KUKA KRL program: EPS_2_251491_MH02A_A_20251118025154.src

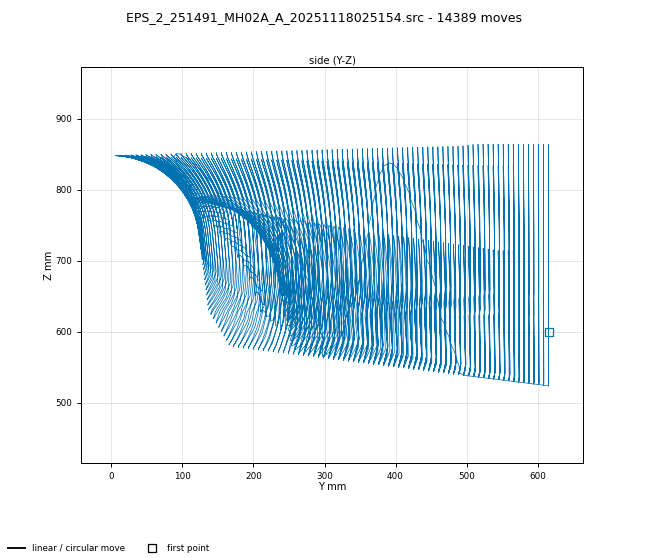
[picture p0: tool path of EPS_2_251491_MH02A_A_20251118025154.src, 14389 of 14391 moves have a stored position in this frame; points joined in program order, loops and branches not executed]
&ACCESS RVP
&REL 4
&COMMENT QRS 19112012
&PARAM EDITMASK = *
DEF PART()
EXT BAS (BAS_COMMAND :IN,REAL :IN )
INT I
BAS (#INITMOV,0 )

;KUKA QRS Post kuka4.cps  Date:22-06-2017 !

File_ID=2920

QRS_PRE_INIT()

;Init var - Until changes are made in qrs_pre_init
Outlet_Square_prg=0
Inlet_1_Square_prg=0
Inlet_2_Square_prg=0
Inlet_3_Square_prg=0
Inlet_4_Square_prg=0
Inlet_5_Square_prg=0

Outlet_1={X 0.000, Y 513.730, Z 763.500, B 0.000, E1 0.000 }
Inlet_1={X 0.000, Y 515.870, Z 733.500, B 0.000, E1 180.000 }
Inlet_2={X 0.000, Y 545.110, Z 323.500, B 0.000, E1 248.000 }
Outlet_1_type=201
Inlet_1_type=201
Inlet_2_type=201
;QRS#1=Sidecore dimensions
;QRS#2=200-8" PVC SDR 35
;QRS#3=200-8" PVC SDR 35
;QRS#4=200-8" PVC SDR 35
;QRS#5=
;QRS#6=
;QRS#7=
;QRS#8=
;QRS#9=12-08 PSX
;QRS#10=12-08 PSX
;QRS#11=12-08 PSX
;QRS#12=
;QRS#13=
;QRS#14=
;QRS#15=
;QRS#16=1220x127x1143 3,75'
;QRS#17=EPS Height
;QRS#18=864
;QRS#19=*
;QRS#20= UPDATED VERSION 22-06-2017
;QRS#21=*
Outlet_Square=0100
Inlet_1_Square=0100
Inlet_2_Square=0100
Inlet_3_Square=0
Inlet_4_Square=0
Inlet_5_Square=0
Mill_Square=1
Outlet_Square_Prg=204
Inlet_1_Square_prg=204
Inlet_2_Square_prg=204

QRS_INIT()

$ADVANCE=5

; T1
PTP {E1 173.604,E2 173.604}
PTP {X 0,Y 615.506,A -85,B 0,C 180,E1 173.604,E2 173.604,E3 0,E4 0,E5 0,E6 0}
QRS_SPEED_INIT()
LIN {X 0,Y 615.506,Z 600,A -85,B 0,C 180,E1 173.604,E2 173.604,E3 0,E4 0,E5 0,E6 0} C_VEL
LIN {X 0,Y 615.506,Z 533.863,A -85,B 0,C 180,E1 173.604,E2 173.604} C_VEL
LIN {X 0,Y 615.506,Z 525.682,A -85,B 0,C 180,E1 173.604,E2 173.604} C_VEL
LIN {X 0,Y 615.488,Z 523.682,A -85,B 0,C 180,E1 173.418,E2 173.418} C_VEL
LIN {X 0,Y 615.475,Z 523.688,A -85,B 0,C 180,E1 170.801,E2 170.801} C_VEL
LIN {X 0,Y 615.491,Z 523.701,A -85,B 0,C 180,E1 168.139,E2 168.139} C_VEL
LIN {X 0,Y 615.482,Z 523.685,A -85,B 0,C 180,E1 165.451,E2 165.451} C_VEL
LIN {X 0,Y 615.476,Z 523.687,A -85,B 0,C 180,E1 162.729,E2 162.729} C_VEL
LIN {X 0,Y 615.49,Z 523.699,A -85,B 0,C 180,E1 159.967,E2 159.967} C_VEL
LIN {X 0,Y 615.487,Z 523.682,A -85,B 0,C 180,E1 157.155,E2 157.155} C_VEL
LIN {X 0,Y 615.484,Z 523.693,A -85,B 0,C 180,E1 154.284,E2 154.284} C_VEL
LIN {X 0,Y 615.48,Z 523.691,A -85,B 0,C 180,E1 151.551,E2 151.551} C_VEL
LIN {X 0,Y 615.484,Z 523.682,A -85,B 0,C 180,E1 148.914,E2 148.914} C_VEL
LIN {X 0,Y 615.496,Z 523.697,A -85,B 0,C 180,E1 145.978,E2 145.978} C_VEL
LIN {X 0,Y 615.487,Z 523.682,A -85,B 0,C 180,E1 143.063,E2 143.063} C_VEL
LIN {X 0,Y 615.477,Z 523.691,A -85,B 0,C 180,E1 140.249,E2 140.249} C_VEL
LIN {X 0,Y 615.489,Z 523.697,A -85,B 0,C 180,E1 137.647,E2 137.647} C_VEL
LIN {X 0,Y 615.479,Z 523.684,A -85,B 0,C 180,E1 134.93,E2 134.93} C_VEL
LIN {X 0,Y 615.478,Z 523.692,A -85,B 0,C 180,E1 132.079,E2 132.079} C_VEL
LIN {X 0,Y 615.494,Z 523.699,A -85,B 0,C 180,E1 129.75,E2 129.75} C_VEL
LIN {X 0,Y 615.478,Z 523.685,A -85,B 0,C 180,E1 126.935,E2 126.935} C_VEL
LIN {X 0,Y 615.489,Z 523.681,A -85,B 0,C 180,E1 124.7,E2 124.7} C_VEL
LIN {X 0,Y 615.485,Z 523.683,A -85,B 0,C 180,E1 122.33,E2 122.33} C_VEL
LIN {X 0,Y 615.493,Z 523.696,A -85,B 0,C 180,E1 119.406,E2 119.406} C_VEL
LIN {X 0,Y 615.492,Z 523.68,A -85,B 0,C 180,E1 116.444,E2 116.444} C_VEL
LIN {X 0,Y 615.488,Z 523.846,A -85,B 0,C 180,E1 114.239,E2 114.239} C_VEL
LIN {X 0,Y 615.492,Z 547.088,A -85,B 0,C 180,E1 111.432,E2 111.432} C_VEL
LIN {X 0,Y 615.493,Z 570.943,A -85,B 0,C 180,E1 108.605,E2 108.605} C_VEL
LIN {X 0,Y 615.486,Z 594.072,A -85,B 0,C 180,E1 105.906,E2 105.906} C_VEL
LIN {X 0,Y 615.486,Z 618.987,A -85,B 0,C 180,E1 103.034,E2 103.034} C_VEL
LIN {X 0,Y 615.479,Z 620.636,A -85,B 0,C 180,E1 102.845,E2 102.845} C_VEL
LIN {X 0,Y 615.476,Z 729.625,A -85,B 0,C 180,E1 101.548,E2 101.548} C_VEL
LIN {X 0,Y 615.49,Z 742.21,A -85,B 0,C 180,E1 101.277,E2 101.277} C_VEL
LIN {X 0,Y 615.489,Z 755.605,A -85,B 0,C 180,E1 100.842,E2 100.842} C_VEL
LIN {X 0,Y 615.493,Z 766.557,A -85,B 0,C 180,E1 100.361,E2 100.361} C_VEL
LIN {X 0,Y 615.485,Z 778.299,A -85,B 0,C 180,E1 99.697,E2 99.697} C_VEL
LIN {X 0,Y 615.499,Z 788.762,A -85,B 0,C 180,E1 98.951,E2 98.951} C_VEL
LIN {X 0,Y 615.498,Z 797.326,A -85,B 0,C 180,E1 98.206,E2 98.206} C_VEL
LIN {X 0,Y 615.497,Z 805.205,A -85,B 0,C 180,E1 97.381,E2 97.381} C_VEL
LIN {X 0,Y 615.497,Z 812.896,A -85,B 0,C 180,E1 96.392,E2 96.392} C_VEL
LIN {X 0,Y 615.497,Z 819.955,A -85,B 0,C 180,E1 95.242,E2 95.242} C_VEL
LIN {X 0,Y 615.494,Z 824.656,A -85,B 0,C 180,E1 94.257,E2 94.257} C_VEL
LIN {X 0,Y 615.494,Z 828.253,A -85,B 0,C 180,E1 93.273,E2 93.273} C_VEL
LIN {X 0,Y 615.496,Z 830.113,A -85,B 0,C 180,E1 92.618,E2 92.618} C_VEL
LIN {X 0,Y 615.497,Z 831.533,A -85,B 0,C 180,E1 91.964,E2 91.964} C_VEL
LIN {X 0,Y 615.496,Z 833.141,A -85,B 0,C 180,E1 90.655,E2 90.655} C_VEL
LIN {X 0,Y 615.495,Z 833.384,A -85,B 0,C 180,E1 90.001,E2 90.001} C_VEL
LIN {X 0,Y 615.495,Z 833.206,A -85,B 0,C 180,E1 89.346,E2 89.346} C_VEL
LIN {X 0,Y 615.498,Z 831.683,A -85,B 0,C 180,E1 88.038,E2 88.038} C_VEL
LIN {X 0,Y 615.498,Z 830.343,A -85,B 0,C 180,E1 87.383,E2 87.383} C_VEL
LIN {X 0,Y 615.496,Z 827.496,A -85,B 0,C 180,E1 86.4,E2 86.4} C_VEL
LIN {X 0,Y 615.498,Z 823.637,A -85,B 0,C 180,E1 85.416,E2 85.416} C_VEL
LIN {X 0,Y 615.498,Z 818.655,A -85,B 0,C 180,E1 84.431,E2 84.431} C_VEL
LIN {X 0,Y 615.496,Z 812.208,A -85,B 0,C 180,E1 83.418,E2 83.418} C_VEL
LIN {X 0,Y 615.497,Z 804.543,A -85,B 0,C 180,E1 82.455,E2 82.455} C_VEL
LIN {X 0,Y 615.498,Z 794.766,A -85,B 0,C 180,E1 81.464,E2 81.464} C_VEL
LIN {X 0,Y 615.497,Z 784.503,A -85,B 0,C 180,E1 80.636,E2 80.636} C_VEL
LIN {X 0,Y 615.496,Z 772.941,A -85,B 0,C 180,E1 79.89,E2 79.89} C_VEL
LIN {X 0,Y 615.496,Z 761.057,A -85,B 0,C 180,E1 79.292,E2 79.292} C_VEL
LIN {X 0,Y 615.497,Z 748.181,A -85,B 0,C 180,E1 78.808,E2 78.808} C_VEL
LIN {X 0,Y 615.477,Z 735.593,A -85,B 0,C 180,E1 78.474,E2 78.474} C_VEL
LIN {X 0,Y 615.475,Z 722.503,A -85,B 0,C 180,E1 78.265,E2 78.265} C_VEL
LIN {X 0,Y 615.48,Z 621.405,A -85,B 0,C 180,E1 77.072,E2 77.072} C_VEL
LIN {X 0,Y 615.476,Z 599.659,A -85,B 0,C 180,E1 74.265,E2 74.265} C_VEL
LIN {X 0,Y 615.487,Z 578.943,A -85,B 0,C 180,E1 71.56,E2 71.56} C_VEL
LIN {X 0,Y 615.485,Z 557.708,A -85,B 0,C 180,E1 68.745,E2 68.745} C_VEL
LIN {X 0,Y 615.476,Z 537.338,A -85,B 0,C 180,E1 65.995,E2 65.995} C_VEL
LIN {X 0,Y 615.474,Z 523.686,A -85,B 0,C 180,E1 64.103,E2 64.103} C_VEL
LIN {X 0,Y 615.485,Z 523.686,A -85,B 0,C 180,E1 61.343,E2 61.343} C_VEL
LIN {X 0,Y 615.492,Z 523.696,A -85,B 0,C 180,E1 58.914,E2 58.914} C_VEL
LIN {X 0,Y 615.497,Z 523.69,A -85,B 0,C 180,E1 56.465,E2 56.465} C_VEL
LIN {X 0,Y 615.48,Z 523.684,A -85,B 0,C 180,E1 53.576,E2 53.576} C_VEL
LIN {X 0,Y 615.488,Z 523.694,A -85,B 0,C 180,E1 50.938,E2 50.938} C_VEL
LIN {X 0,Y 615.496,Z 523.695,A -85,B 0,C 180,E1 48.528,E2 48.528} C_VEL
LIN {X 0,Y 615.477,Z 523.685,A -85,B 0,C 180,E1 45.851,E2 45.851} C_VEL
LIN {X 0,Y 615.493,Z 523.688,A -85,B 0,C 180,E1 43.05,E2 43.05} C_VEL
LIN {X 0,Y 615.493,Z 523.685,A -85,B 0,C 180,E1 40.092,E2 40.092} C_VEL
LIN {X 0,Y 615.489,Z 523.684,A -85,B 0,C 180,E1 37.242,E2 37.242} C_VEL
LIN {X 0,Y 615.497,Z 523.701,A -85,B 0,C 180,E1 34.575,E2 34.575} C_VEL
LIN {X 0,Y 615.474,Z 610.382,A -85,B 0,C 180,E1 33.535,E2 33.535} C_VEL
LIN {X 0,Y 615.48,Z 623.669,A -85,B 0,C 180,E1 33.237,E2 33.237} C_VEL
LIN {X 0,Y 615.494,Z 636.803,A -85,B 0,C 180,E1 32.797,E2 32.797} C_VEL
LIN {X 0,Y 615.482,Z 648.688,A -85,B 0,C 180,E1 32.251,E2 32.251} C_VEL
LIN {X 0,Y 615.486,Z 660.755,A -85,B 0,C 180,E1 31.536,E2 31.536} C_VEL
LIN {X 0,Y 615.497,Z 671.49,A -85,B 0,C 180,E1 30.729,E2 30.729} C_VEL
LIN {X 0,Y 615.499,Z 681.399,A -85,B 0,C 180,E1 29.799,E2 29.799} C_VEL
LIN {X 0,Y 615.497,Z 689.587,A -85,B 0,C 180,E1 28.844,E2 28.844} C_VEL
LIN {X 0,Y 615.493,Z 697.177,A -85,B 0,C 180,E1 27.73,E2 27.73} C_VEL
LIN {X 0,Y 615.493,Z 702.466,A -85,B 0,C 180,E1 26.746,E2 26.746} C_VEL
LIN {X 0,Y 615.496,Z 707.29,A -85,B 0,C 180,E1 25.573,E2 25.573} C_VEL
LIN {X 0,Y 615.493,Z 709.114,A -85,B 0,C 180,E1 24.992,E2 24.992} C_VEL
LIN {X 0,Y 615.494,Z 711.448,A -85,B 0,C 180,E1 24.013,E2 24.013} C_VEL
LIN {X 0,Y 615.496,Z 713.008,A -85,B 0,C 180,E1 22.844,E2 22.844} C_VEL
LIN {X 0,Y 615.495,Z 713.351,A -85,B 0,C 180,E1 22.136,E2 22.136} C_VEL
LIN {X 0,Y 615.497,Z 713.263,A -85,B 0,C 180,E1 21.432,E2 21.432} C_VEL
LIN {X 0,Y 615.495,Z 712.482,A -85,B 0,C 180,E1 20.563,E2 20.563} C_VEL
LIN {X 0,Y 615.494,Z 710.235,A -85,B 0,C 180,E1 19.338,E2 19.338} C_VEL
LIN {X 0,Y 615.497,Z 707.103,A -85,B 0,C 180,E1 18.284,E2 18.284} C_VEL
LIN {X 0,Y 615.496,Z 702.986,A -85,B 0,C 180,E1 17.27,E2 17.27} C_VEL
LIN {X 0,Y 615.497,Z 697.127,A -85,B 0,C 180,E1 16.172,E2 16.172} C_VEL
LIN {X 0,Y 615.496,Z 689.518,A -85,B 0,C 180,E1 15.056,E2 15.056} C_VEL
LIN {X 0,Y 615.498,Z 681.234,A -85,B 0,C 180,E1 14.094,E2 14.094} C_VEL
LIN {X 0,Y 615.499,Z 671.722,A -85,B 0,C 180,E1 13.201,E2 13.201} C_VEL
LIN {X 0,Y 615.486,Z 661.855,A -85,B 0,C 180,E1 12.446,E2 12.446} C_VEL
LIN {X 0,Y 615.492,Z 650.912,A -85,B 0,C 180,E1 11.777,E2 11.777} C_VEL
LIN {X 0,Y 615.491,Z 638.717,A -85,B 0,C 180,E1 11.193,E2 11.193} C_VEL
LIN {X 0,Y 615.495,Z 626.639,A -85,B 0,C 180,E1 10.758,E2 10.758} C_VEL
LIN {X 0,Y 615.483,Z 614.11,A -85,B 0,C 180,E1 10.444,E2 10.444} C_VEL
LIN {X 0,Y 615.476,Z 598.256,A -85,B 0,C 180,E1 10.215,E2 10.215} C_VEL
LIN {X 0,Y 615.493,Z 523.77,A -85,B 0,C 180,E1 9.344,E2 9.344} C_VEL
LIN {X 0,Y 615.489,Z 523.682,A -85,B 0,C 180,E1 6.557,E2 6.557} C_VEL
LIN {X 0,Y 615.477,Z 523.687,A -85,B 0,C 180,E1 3.929,E2 3.929} C_VEL
LIN {X 0,Y 615.496,Z 523.701,A -85,B 0,C 180,E1 1.309,E2 1.309} C_VEL
LIN {X 0,Y 615.488,Z 523.685,A -85,B 0,C 180,E1 -1.309,E2 -1.309} C_VEL
LIN {X 0,Y 615.478,Z 523.685,A -85,B 0,C 180,E1 -3.929,E2 -3.929} C_VEL
LIN {X 0,Y 615.489,Z 523.698,A -85,B 0,C 180,E1 -6.592,E2 -6.592} C_VEL
LIN {X 0,Y 615.479,Z 523.689,A -85,B 0,C 180,E1 -9.199,E2 -9.199} C_VEL
LIN {X 0,Y 615.485,Z 523.682,A -85,B 0,C 180,E1 -11.861,E2 -11.861} C_VEL
LIN {X 0,Y 615.48,Z 523.697,A -85,B 0,C 180,E1 -14.549,E2 -14.549} C_VEL
LIN {X 0,Y 615.476,Z 523.689,A -85,B 0,C 180,E1 -17.271,E2 -17.271} C_VEL
LIN {X 0,Y 615.486,Z 523.684,A -85,B 0,C 180,E1 -20.033,E2 -20.033} C_VEL
LIN {X 0,Y 615.492,Z 523.699,A -85,B 0,C 180,E1 -22.844,E2 -22.844} C_VEL
LIN {X 0,Y 615.484,Z 523.682,A -85,B 0,C 180,E1 -25.716,E2 -25.716} C_VEL
LIN {X 0,Y 615.485,Z 523.692,A -85,B 0,C 180,E1 -28.453,E2 -28.453} C_VEL
LIN {X 0,Y 615.487,Z 523.692,A -85,B 0,C 180,E1 -31.088,E2 -31.088} C_VEL
LIN {X 0,Y 615.496,Z 523.681,A -85,B 0,C 180,E1 -34.022,E2 -34.022} C_VEL
LIN {X 0,Y 615.494,Z 523.697,A -85,B 0,C 180,E1 -36.94,E2 -36.94} C_VEL
LIN {X 0,Y 615.475,Z 523.685,A -85,B 0,C 180,E1 -39.751,E2 -39.751} C_VEL
LIN {X 0,Y 615.493,Z 523.686,A -85,B 0,C 180,E1 -42.353,E2 -42.353} C_VEL
LIN {X 0,Y 615.492,Z 523.694,A -85,B 0,C 180,E1 -45.068,E2 -45.068} C_VEL
LIN {X 0,Y 615.477,Z 523.684,A -85,B 0,C 180,E1 -47.921,E2 -47.921} C_VEL
LIN {X 0,Y 615.493,Z 523.684,A -85,B 0,C 180,E1 -50.252,E2 -50.252} C_VEL
LIN {X 0,Y 615.491,Z 523.695,A -85,B 0,C 180,E1 -53.063,E2 -53.063} C_VEL
LIN {X 0,Y 615.49,Z 523.688,A -85,B 0,C 180,E1 -55.299,E2 -55.299} C_VEL
LIN {X 0,Y 615.484,Z 523.683,A -85,B 0,C 180,E1 -57.67,E2 -57.67} C_VEL
LIN {X 0,Y 615.498,Z 523.69,A -85,B 0,C 180,E1 -60.595,E2 -60.595} C_VEL
LIN {X 0,Y 615.491,Z 523.683,A -85,B 0,C 180,E1 -63.557,E2 -63.557} C_VEL
LIN {X 0,Y 615.474,Z 523.886,A -85,B 0,C 180,E1 -64.08,E2 -64.08} C_VEL
LIN {X 0,Y 615.484,Z 549.311,A -85,B 0,C 180,E1 -66.801,E2 -66.801} C_VEL
LIN {X 0,Y 615.487,Z 575.784,A -85,B 0,C 180,E1 -69.576,E2 -69.576} C_VEL
LIN {X 0,Y 615.49,Z 603.095,A -85,B 0,C 180,E1 -72.388,E2 -72.388} C_VEL
LIN {X 0,Y 615.481,Z 629.946,A -85,B 0,C 180,E1 -75.113,E2 -75.113} C_VEL
LIN {X 0,Y 615.488,Z 649.643,A -85,B 0,C 180,E1 -77.093,E2 -77.093} C_VEL
LIN {X 0,Y 615.476,Z 759.874,A -85,B 0,C 180,E1 -78.411,E2 -78.411} C_VEL
LIN {X 0,Y 615.487,Z 772.371,A -85,B 0,C 180,E1 -78.683,E2 -78.683} C_VEL
LIN {X 0,Y 615.496,Z 785.511,A -85,B 0,C 180,E1 -79.109,E2 -79.109} C_VEL
LIN {X 0,Y 615.484,Z 797.491,A -85,B 0,C 180,E1 -79.64,E2 -79.64} C_VEL
LIN {X 0,Y 615.483,Z 809.007,A -85,B 0,C 180,E1 -80.304,E2 -80.304} C_VEL
LIN {X 0,Y 615.499,Z 819.35,A -85,B 0,C 180,E1 -81.051,E2 -81.051} C_VEL
LIN {X 0,Y 615.497,Z 827.819,A -85,B 0,C 180,E1 -81.795,E2 -81.795} C_VEL
LIN {X 0,Y 615.498,Z 835.612,A -85,B 0,C 180,E1 -82.62,E2 -82.62} C_VEL
LIN {X 0,Y 615.496,Z 843.207,A -85,B 0,C 180,E1 -83.609,E2 -83.609} C_VEL
LIN {X 0,Y 615.498,Z 850.208,A -85,B 0,C 180,E1 -84.76,E2 -84.76} C_VEL
LIN {X 0,Y 615.494,Z 854.854,A -85,B 0,C 180,E1 -85.744,E2 -85.744} C_VEL
LIN {X 0,Y 615.496,Z 858.4,A -85,B 0,C 180,E1 -86.728,E2 -86.728} C_VEL
LIN {X 0,Y 615.497,Z 860.234,A -85,B 0,C 180,E1 -87.383,E2 -87.383} C_VEL
LIN {X 0,Y 615.496,Z 861.609,A -85,B 0,C 180,E1 -88.038,E2 -88.038} C_VEL
LIN {X 0,Y 615.496,Z 863.174,A -85,B 0,C 180,E1 -89.346,E2 -89.346} C_VEL
LIN {X 0,Y 615.494,Z 863.389,A -85,B 0,C 180,E1 -90.001,E2 -90.001} C_VEL
LIN {X 0,Y 615.496,Z 862.579,A -85,B 0,C 180,E1 -91.309,E2 -91.309} C_VEL
LIN {X 0,Y 615.496,Z 861.607,A -85,B 0,C 180,E1 -91.964,E2 -91.964} C_VEL
LIN {X 0,Y 615.497,Z 860.232,A -85,B 0,C 180,E1 -92.618,E2 -92.618} C_VEL
LIN {X 0,Y 615.496,Z 857.348,A -85,B 0,C 180,E1 -93.601,E2 -93.601} C_VEL
LIN {X 0,Y 615.498,Z 853.439,A -85,B 0,C 180,E1 -94.585,E2 -94.585} C_VEL
LIN {X 0,Y 615.499,Z 848.402,A -85,B 0,C 180,E1 -95.57,E2 -95.57} C_VEL
LIN {X 0,Y 615.497,Z 841.869,A -85,B 0,C 180,E1 -96.583,E2 -96.583} C_VEL
LIN {X 0,Y 615.497,Z 834.129,A -85,B 0,C 180,E1 -97.546,E2 -97.546} C_VEL
LIN {X 0,Y 615.498,Z 826.04,A -85,B 0,C 180,E1 -98.372,E2 -98.372} C_VEL
LIN {X 0,Y 615.499,Z 816.162,A -85,B 0,C 180,E1 -99.199,E2 -99.199} C_VEL
LIN {X 0,Y 615.486,Z 804.975,A -85,B 0,C 180,E1 -99.946,E2 -99.946} C_VEL
LIN {X 0,Y 615.483,Z 794.015,A -85,B 0,C 180,E1 -100.527,E2 -100.527} C_VEL
LIN {X 0,Y 615.496,Z 781.425,A -85,B 0,C 180,E1 -101.042,E2 -101.042} C_VEL
LIN {X 0,Y 615.482,Z 769.049,A -85,B 0,C 180,E1 -101.402,E2 -101.402} C_VEL
LIN {X 0,Y 615.475,Z 755.442,A -85,B 0,C 180,E1 -101.653,E2 -101.653} C_VEL
LIN {X 0,Y 615.493,Z 650.529,A -85,B 0,C 180,E1 -102.887,E2 -102.887} C_VEL
LIN {X 0,Y 615.496,Z 625.281,A -85,B 0,C 180,E1 -105.735,E2 -105.735} C_VEL
LIN {X 0,Y 615.488,Z 601.591,A -85,B 0,C 180,E1 -108.441,E2 -108.441} C_VEL
LIN {X 0,Y 615.491,Z 577.301,A -85,B 0,C 180,E1 -111.256,E2 -111.256} C_VEL
LIN {X 0,Y 615.486,Z 554.004,A -85,B 0,C 180,E1 -114.007,E2 -114.007} C_VEL
LIN {X 0,Y 615.492,Z 531.309,A -85,B 0,C 180,E1 -116.745,E2 -116.745} C_VEL
LIN {X 0,Y 615.483,Z 523.683,A -85,B 0,C 180,E1 -117.684,E2 -117.684} C_VEL
LIN {X 0,Y 615.477,Z 523.685,A -85,B 0,C 180,E1 -120.161,E2 -120.161} C_VEL
LIN {X 0,Y 615.487,Z 523.687,A -85,B 0,C 180,E1 -122.458,E2 -122.458} C_VEL
LIN {X 0,Y 615.491,Z 523.695,A -85,B 0,C 180,E1 -124.815,E2 -124.815} C_VEL
LIN {X 0,Y 615.491,Z 523.694,A -85,B 0,C 180,E1 -127.242,E2 -127.242} C_VEL
LIN {X 0,Y 615.477,Z 523.684,A -85,B 0,C 180,E1 -130.088,E2 -130.088} C_VEL
LIN {X 0,Y 615.478,Z 523.685,A -85,B 0,C 180,E1 -132.354,E2 -132.354} C_VEL
LIN {X 0,Y 615.492,Z 523.7,A -85,B 0,C 180,E1 -135.068,E2 -135.068} C_VEL
LIN {X 0,Y 615.49,Z 523.682,A -85,B 0,C 180,E1 -137.919,E2 -137.919} C_VEL
LIN {X 0,Y 615.475,Z 523.684,A -85,B 0,C 180,E1 -140.249,E2 -140.249} C_VEL
LIN {X 0,Y 615.494,Z 523.695,A -85,B 0,C 180,E1 -143.062,E2 -143.062} C_VEL
LIN {X 0,Y 615.495,Z 523.681,A -85,B 0,C 180,E1 -145.978,E2 -145.978} C_VEL
LIN {X 0,Y 615.478,Z 523.683,A -85,B 0,C 180,E1 -148.314,E2 -148.314} C_VEL
LIN {X 0,Y 615.477,Z 523.685,A -85,B 0,C 180,E1 -150.593,E2 -150.593} C_VEL
LIN {X 0,Y 615.489,Z 523.689,A -85,B 0,C 180,E1 -152.954,E2 -152.954} C_VEL
LIN {X 0,Y 615.485,Z 523.691,A -85,B 0,C 180,E1 -155.728,E2 -155.728} C_VEL
LIN {X 0,Y 615.488,Z 523.688,A -85,B 0,C 180,E1 -157.864,E2 -157.864} C_VEL
LIN {X 0,Y 615.476,Z 523.685,A -85,B 0,C 180,E1 -160.662,E2 -160.662} C_VEL
LIN {X 0,Y 615.495,Z 523.699,A -85,B 0,C 180,E1 -163.414,E2 -163.414} C_VEL
LIN {X 0,Y 615.492,Z 523.684,A -85,B 0,C 180,E1 -166.126,E2 -166.126} C_VEL
LIN {X 0,Y 615.476,Z 523.685,A -85,B 0,C 180,E1 -168.807,E2 -168.807} C_VEL
LIN {X 0,Y 615.496,Z 523.696,A -85,B 0,C 180,E1 -171.463,E2 -171.463} C_VEL
LIN {X 0,Y 615.485,Z 523.687,A -85,B 0,C 180,E1 -174.101,E2 -174.101} C_VEL
LIN {X 0,Y 615.481,Z 523.683,A -85,B 0,C 180,E1 -176.727,E2 -176.727} C_VEL
LIN {X 0,Y 615.483,Z 523.692,A -85,B 0,C 180,E1 -179.346,E2 -179.346} C_VEL
LIN {X 0,Y 615.482,Z 523.695,A -85,B 0,C 180,E1 -181.963,E2 -181.963} C_VEL
LIN {X 0,Y 615.498,Z 523.679,A -85,B 0,C 180,E1 -184.585,E2 -184.585} C_VEL
LIN {X 0,Y 615.488,Z 523.682,A -85,B 0,C 180,E1 -186.582,E2 -186.582} C_VEL
LIN {X 0,Y 614.804,Z 523.835,A -85,B 0,C 180,E1 -187.128,E2 -187.128} C_VEL
LIN {X 0,Y 611.96,Z 524.257,A -85,B 0,C 180,E1 -188.014,E2 -188.014} C_VEL
LIN {X 0,Y 609.57,Z 524.564,A -85,B 0,C 180,E1 -188.726,E2 -188.726} C_VEL
LIN {X 0,Y 608.541,Z 524.68,A -85,B 0,C 180,E1 -189.276,E2 -189.276} C_VEL
LIN {X 0,Y 608.456,Z 524.69,A -85,B 0,C 180,E1 -189.462,E2 -189.462} C_VEL
LIN {X 0,Y 608.466,Z 524.693,A -85,B 0,C 180,E1 -192,E2 -192} C_VEL
LIN {X 0,Y 608.47,Z 524.685,A -85,B 0,C 180,E1 -194.721,E2 -194.721} C_VEL
LIN {X 0,Y 608.449,Z 524.691,A -85,B 0,C 180,E1 -197.477,E2 -197.477} C_VEL
LIN {X 0,Y 608.463,Z 524.691,A -85,B 0,C 180,E1 -200.274,E2 -200.274} C_VEL
LIN {X 0,Y 608.448,Z 524.688,A -85,B 0,C 180,E1 -203.124,E2 -203.124} C_VEL
LIN {X 0,Y 608.468,Z 524.691,A -85,B 0,C 180,E1 -205.721,E2 -205.721} C_VEL
LIN {X 0,Y 608.448,Z 524.694,A -85,B 0,C 180,E1 -208.267,E2 -208.267} C_VEL
LIN {X 0,Y 608.474,Z 524.687,A -85,B 0,C 180,E1 -210.545,E2 -210.545} C_VEL
LIN {X 0,Y 608.453,Z 524.687,A -85,B 0,C 180,E1 -212.88,E2 -212.88} C_VEL
LIN {X 0,Y 608.434,Z 524.689,A -85,B 0,C 180,E1 -215.279,E2 -215.279} C_VEL
LIN {X 0,Y 608.472,Z 524.688,A -85,B 0,C 180,E1 -217.746,E2 -217.746} C_VEL
LIN {X 0,Y 608.452,Z 524.696,A -85,B 0,C 180,E1 -220.329,E2 -220.329} C_VEL
LIN {X 0,Y 608.484,Z 524.683,A -85,B 0,C 180,E1 -223.31,E2 -223.31} C_VEL
LIN {X 0,Y 608.466,Z 524.694,A -85,B 0,C 180,E1 -226.13,E2 -226.13} C_VEL
LIN {X 0,Y 608.447,Z 524.69,A -85,B 0,C 180,E1 -228.823,E2 -228.823} C_VEL
LIN {X 0,Y 608.461,Z 524.688,A -85,B 0,C 180,E1 -231.761,E2 -231.761} C_VEL
LIN {X 0,Y 608.449,Z 524.691,A -85,B 0,C 180,E1 -233.955,E2 -233.955} C_VEL
LIN {X 0,Y 608.467,Z 524.695,A -85,B 0,C 180,E1 -236.329,E2 -236.329} C_VEL
LIN {X 0,Y 608.446,Z 524.693,A -85,B 0,C 180,E1 -238.733,E2 -238.733} C_VEL
LIN {X 0,Y 608.474,Z 524.684,A -85,B 0,C 180,E1 -241.38,E2 -241.38} C_VEL
LIN {X 0,Y 608.475,Z 524.692,A -85,B 0,C 180,E1 -244.279,E2 -244.279} C_VEL
LIN {X 0,Y 608.494,Z 524.843,A -85,B 0,C 180,E1 -245.587,E2 -245.587} C_VEL
LIN {X 0,Y 608.637,Z 540.255,A -85,B 0,C 180,E1 -247.484,E2 -247.484} C_VEL
LIN {X 0,Y 608.566,Z 564.729,A -85,B 0,C 180,E1 -250.433,E2 -250.433} C_VEL
LIN {X 0,Y 608.532,Z 586.776,A -85,B 0,C 180,E1 -253.045,E2 -253.045} C_VEL
LIN {X 0,Y 608.511,Z 610.293,A -85,B 0,C 180,E1 -255.793,E2 -255.793} C_VEL
LIN {X 0,Y 608.489,Z 621.002,A -85,B 0,C 180,E1 -257.015,E2 -257.015} C_VEL
LIN {X 0,Y 608.539,Z 729.77,A -85,B 0,C 180,E1 -258.318,E2 -258.318} C_VEL
LIN {X 0,Y 608.528,Z 743.106,A -85,B 0,C 180,E1 -258.614,E2 -258.614} C_VEL
LIN {X 0,Y 608.523,Z 756.433,A -85,B 0,C 180,E1 -259.058,E2 -259.058} C_VEL
LIN {X 0,Y 608.503,Z 768.363,A -85,B 0,C 180,E1 -259.603,E2 -259.603} C_VEL
LIN {X 0,Y 608.498,Z 779.784,A -85,B 0,C 180,E1 -260.275,E2 -260.275} C_VEL
LIN {X 0,Y 608.474,Z 790.079,A -85,B 0,C 180,E1 -261.029,E2 -261.029} C_VEL
LIN {X 0,Y 608.464,Z 799.347,A -85,B 0,C 180,E1 -261.865,E2 -261.865} C_VEL
LIN {X 0,Y 608.467,Z 808.32,A -85,B 0,C 180,E1 -262.867,E2 -262.867} C_VEL
LIN {X 0,Y 608.444,Z 815.552,A -85,B 0,C 180,E1 -263.866,E2 -263.866} C_VEL
LIN {X 0,Y 608.462,Z 820.432,A -85,B 0,C 180,E1 -264.698,E2 -264.698} C_VEL
LIN {X 0,Y 608.439,Z 825.176,A -85,B 0,C 180,E1 -265.694,E2 -265.694} C_VEL
LIN {X 0,Y 608.425,Z 828.811,A -85,B 0,C 180,E1 -266.689,E2 -266.689} C_VEL
LIN {X 0,Y 608.425,Z 830.689,A -85,B 0,C 180,E1 -267.351,E2 -267.351} C_VEL
LIN {X 0,Y 608.443,Z 832.126,A -85,B 0,C 180,E1 -268.014,E2 -268.014} C_VEL
LIN {X 0,Y 608.439,Z 833.751,A -85,B 0,C 180,E1 -269.338,E2 -269.338} C_VEL
LIN {X 0,Y 608.435,Z 833.995,A -85,B 0,C 180,E1 -269.999,E2 -269.999} C_VEL
LIN {X 0,Y 608.438,Z 833.815,A -85,B 0,C 180,E1 -270.661,E2 -270.661} C_VEL
LIN {X 0,Y 608.443,Z 832.277,A -85,B 0,C 180,E1 -271.985,E2 -271.985} C_VEL
LIN {X 0,Y 608.426,Z 830.92,A -85,B 0,C 180,E1 -272.648,E2 -272.648} C_VEL
LIN {X 0,Y 608.449,Z 828.044,A -85,B 0,C 180,E1 -273.642,E2 -273.642} C_VEL
LIN {X 0,Y 608.433,Z 824.146,A -85,B 0,C 180,E1 -274.637,E2 -274.637} C_VEL
LIN {X 0,Y 608.449,Z 819.116,A -85,B 0,C 180,E1 -275.634,E2 -275.634} C_VEL
LIN {X 0,Y 608.441,Z 812.799,A -85,B 0,C 180,E1 -276.632,E2 -276.632} C_VEL
LIN {X 0,Y 608.475,Z 804.885,A -85,B 0,C 180,E1 -277.632,E2 -277.632} C_VEL
LIN {X 0,Y 608.472,Z 795.044,A -85,B 0,C 180,E1 -278.635,E2 -278.635} C_VEL
LIN {X 0,Y 608.479,Z 784.724,A -85,B 0,C 180,E1 -279.473,E2 -279.473} C_VEL
LIN {X 0,Y 608.494,Z 773.113,A -85,B 0,C 180,E1 -280.228,E2 -280.228} C_VEL
LIN {X 0,Y 608.519,Z 760.879,A -85,B 0,C 180,E1 -280.845,E2 -280.845} C_VEL
LIN {X 0,Y 608.525,Z 748.288,A -85,B 0,C 180,E1 -281.322,E2 -281.322} C_VEL
LIN {X 0,Y 608.529,Z 735.684,A -85,B 0,C 180,E1 -281.66,E2 -281.66} C_VEL
LIN {X 0,Y 608.535,Z 722.605,A -85,B 0,C 180,E1 -281.871,E2 -281.871} C_VEL
LIN {X 0,Y 608.476,Z 621.548,A -85,B 0,C 180,E1 -283.079,E2 -283.079} C_VEL
LIN {X 0,Y 608.486,Z 601.034,A -85,B 0,C 180,E1 -285.748,E2 -285.748} C_VEL
LIN {X 0,Y 608.549,Z 580.194,A -85,B 0,C 180,E1 -288.494,E2 -288.494} C_VEL
LIN {X 0,Y 608.568,Z 559.018,A -85,B 0,C 180,E1 -291.331,E2 -291.331} C_VEL
LIN {X 0,Y 608.597,Z 538.182,A -85,B 0,C 180,E1 -294.177,E2 -294.177} C_VEL
LIN {X 0,Y 608.485,Z 524.878,A -85,B 0,C 180,E1 -296.033,E2 -296.033} C_VEL
LIN {X 0,Y 608.476,Z 524.686,A -85,B 0,C 180,E1 -298.62,E2 -298.62} C_VEL
LIN {X 0,Y 608.477,Z 524.694,A -85,B 0,C 180,E1 -301.315,E2 -301.315} C_VEL
LIN {X 0,Y 608.476,Z 524.687,A -85,B 0,C 180,E1 -303.735,E2 -303.735} C_VEL
LIN {X 0,Y 608.473,Z 524.685,A -85,B 0,C 180,E1 -306.089,E2 -306.089} C_VEL
LIN {X 0,Y 608.467,Z 524.686,A -85,B 0,C 180,E1 -308.587,E2 -308.587} C_VEL
LIN {X 0,Y 608.469,Z 524.696,A -85,B 0,C 180,E1 -311.343,E2 -311.343} C_VEL
LIN {X 0,Y 608.448,Z 524.687,A -85,B 0,C 180,E1 -314.263,E2 -314.263} C_VEL
LIN {X 0,Y 608.459,Z 524.691,A -85,B 0,C 180,E1 -317.04,E2 -317.04} C_VEL
LIN {X 0,Y 608.459,Z 524.692,A -85,B 0,C 180,E1 -319.697,E2 -319.697} C_VEL
LIN {X 0,Y 608.469,Z 524.685,A -85,B 0,C 180,E1 -322.254,E2 -322.254} C_VEL
LIN {X 0,Y 608.477,Z 524.691,A -85,B 0,C 180,E1 -325.185,E2 -325.185} C_VEL
LIN {X 0,Y 608.508,Z 524.897,A -85,B 0,C 180,E1 -325.299,E2 -325.299} C_VEL
LIN {X 0,Y 608.52,Z 610.577,A -85,B 0,C 180,E1 -326.333,E2 -326.333} C_VEL
LIN {X 0,Y 608.531,Z 624.178,A -85,B 0,C 180,E1 -326.643,E2 -326.643} C_VEL
LIN {X 0,Y 608.515,Z 636.869,A -85,B 0,C 180,E1 -327.075,E2 -327.075} C_VEL
LIN {X 0,Y 608.492,Z 649.44,A -85,B 0,C 180,E1 -327.661,E2 -327.661} C_VEL
LIN {X 0,Y 608.485,Z 660.108,A -85,B 0,C 180,E1 -328.296,E2 -328.296} C_VEL
LIN {X 0,Y 608.496,Z 670.606,A -85,B 0,C 180,E1 -329.071,E2 -329.071} C_VEL
LIN {X 0,Y 608.458,Z 680.144,A -85,B 0,C 180,E1 -329.947,E2 -329.947} C_VEL
LIN {X 0,Y 608.458,Z 689.233,A -85,B 0,C 180,E1 -330.979,E2 -330.979} C_VEL
LIN {X 0,Y 608.449,Z 695.905,A -85,B 0,C 180,E1 -331.921,E2 -331.921} C_VEL
LIN {X 0,Y 608.439,Z 702.059,A -85,B 0,C 180,E1 -333.012,E2 -333.012} C_VEL
LIN {X 0,Y 608.431,Z 706.278,A -85,B 0,C 180,E1 -333.964,E2 -333.964} C_VEL
LIN {X 0,Y 608.427,Z 709.921,A -85,B 0,C 180,E1 -335.063,E2 -335.063} C_VEL
LIN {X 0,Y 608.439,Z 712.359,A -85,B 0,C 180,E1 -336.154,E2 -336.154} C_VEL
LIN {X 0,Y 608.431,Z 713.365,A -85,B 0,C 180,E1 -336.875,E2 -336.875} C_VEL
LIN {X 0,Y 608.423,Z 713.9,A -85,B 0,C 180,E1 -337.593,E2 -337.593} C_VEL
LIN {X 0,Y 608.416,Z 713.945,A -85,B 0,C 180,E1 -338.306,E2 -338.306} C_VEL
LIN {X 0,Y 608.438,Z 713.235,A -85,B 0,C 180,E1 -339.325,E2 -339.325} C_VEL
LIN {X 0,Y 608.416,Z 711.397,A -85,B 0,C 180,E1 -340.428,E2 -340.428} C_VEL
LIN {X 0,Y 608.425,Z 709.157,A -85,B 0,C 180,E1 -341.292,E2 -341.292} C_VEL
LIN {X 0,Y 608.428,Z 704.634,A -85,B 0,C 180,E1 -342.523,E2 -342.523} C_VEL
LIN {X 0,Y 608.438,Z 698.8,A -85,B 0,C 180,E1 -343.691,E2 -343.691} C_VEL
LIN {X 0,Y 608.456,Z 691.824,A -85,B 0,C 180,E1 -344.765,E2 -344.765} C_VEL
LIN {X 0,Y 608.457,Z 683.467,A -85,B 0,C 180,E1 -345.792,E2 -345.792} C_VEL
LIN {X 0,Y 608.481,Z 674.939,A -85,B 0,C 180,E1 -346.644,E2 -346.644} C_VEL
LIN {X 0,Y 608.487,Z 664.445,A -85,B 0,C 180,E1 -347.493,E2 -347.493} C_VEL
LIN {X 0,Y 608.498,Z 652.664,A -85,B 0,C 180,E1 -348.254,E2 -348.254} C_VEL
LIN {X 0,Y 608.524,Z 640.279,A -85,B 0,C 180,E1 -348.87,E2 -348.87} C_VEL
LIN {X 0,Y 608.541,Z 628.798,A -85,B 0,C 180,E1 -349.305,E2 -349.305} C_VEL
LIN {X 0,Y 608.526,Z 616.282,A -85,B 0,C 180,E1 -349.646,E2 -349.646} C_VEL
LIN {X 0,Y 608.531,Z 603.871,A -85,B 0,C 180,E1 -349.856,E2 -349.856} C_VEL
LIN {X 0,Y 608.487,Z 524.691,A -85,B 0,C 180,E1 -350.799,E2 -350.799} C_VEL
LIN {X 0,Y 608.465,Z 524.687,A -85,B 0,C 180,E1 -353.367,E2 -353.367} C_VEL
LIN {X 0,Y 608.448,Z 524.689,A -85,B 0,C 180,E1 -356.026,E2 -356.026} C_VEL
LIN {X 0,Y 608.477,Z 524.695,A -85,B 0,C 180,E1 -358.676,E2 -358.676} C_VEL
LIN {X 0,Y 608.47,Z 524.686,A -85,B 0,C 180,E1 -361.324,E2 -361.324} C_VEL
LIN {X 0,Y 608.448,Z 524.688,A -85,B 0,C 180,E1 -363.974,E2 -363.974} C_VEL
LIN {X 0,Y 608.465,Z 524.695,A -85,B 0,C 180,E1 -366.633,E2 -366.633} C_VEL
LIN {X 0,Y 608.464,Z 524.688,A -85,B 0,C 180,E1 -369.306,E2 -369.306} C_VEL
LIN {X 0,Y 608.46,Z 524.687,A -85,B 0,C 180,E1 -372,E2 -372} C_VEL
LIN {X 0,Y 608.467,Z 524.696,A -85,B 0,C 180,E1 -374.721,E2 -374.721} C_VEL
LIN {X 0,Y 608.446,Z 524.689,A -85,B 0,C 180,E1 -377.477,E2 -377.477} C_VEL
LIN {X 0,Y 608.461,Z 524.689,A -85,B 0,C 180,E1 -380.274,E2 -380.274} C_VEL
LIN {X 0,Y 608.45,Z 524.692,A -85,B 0,C 180,E1 -383.124,E2 -383.124} C_VEL
LIN {X 0,Y 608.466,Z 524.685,A -85,B 0,C 180,E1 -385.723,E2 -385.723} C_VEL
LIN {X 0,Y 608.474,Z 524.692,A -85,B 0,C 180,E1 -388.623,E2 -388.623} C_VEL
LIN {X 0,Y 608.47,Z 524.688,A -85,B 0,C 180,E1 -391.316,E2 -391.316} C_VEL
LIN {X 0,Y 608.468,Z 524.685,A -85,B 0,C 180,E1 -393.737,E2 -393.737} C_VEL
LIN {X 0,Y 608.47,Z 524.686,A -85,B 0,C 180,E1 -396.091,E2 -396.091} C_VEL
LIN {X 0,Y 608.475,Z 524.691,A -85,B 0,C 180,E1 -398.588,E2 -398.588} C_VEL
LIN {X 0,Y 608.46,Z 524.689,A -85,B 0,C 180,E1 -401.344,E2 -401.344} C_VEL
LIN {X 0,Y 608.461,Z 524.688,A -85,B 0,C 180,E1 -404.266,E2 -404.266} C_VEL
LIN {X 0,Y 608.456,Z 524.694,A -85,B 0,C 180,E1 -407.042,E2 -407.042} C_VEL
LIN {X 0,Y 608.447,Z 524.688,A -85,B 0,C 180,E1 -409.698,E2 -409.698} C_VEL
LIN {X 0,Y 608.466,Z 524.687,A -85,B 0,C 180,E1 -412.255,E2 -412.255} C_VEL
LIN {X 0,Y 608.476,Z 524.691,A -85,B 0,C 180,E1 -415.091,E2 -415.091} C_VEL
LIN {X 0,Y 608.466,Z 524.685,A -85,B 0,C 180,E1 -417.907,E2 -417.907} C_VEL
LIN {X 0,Y 608.463,Z 524.687,A -85,B 0,C 180,E1 -420.221,E2 -420.221} C_VEL
LIN {X 0,Y 608.487,Z 524.692,A -85,B 0,C 180,E1 -422.792,E2 -422.792} C_VEL
LIN {X 0,Y 608.474,Z 524.727,A -85,B 0,C 180,E1 -423.852,E2 -423.852} C_VEL
LIN {X 0,Y 608.716,Z 528.099,A -85,B 0,C 180,E1 -424.232,E2 -424.232} C_VEL
LIN {X 0,Y 608.654,Z 552.673,A -85,B 0,C 180,E1 -426.885,E2 -426.885} C_VEL
LIN {X 0,Y 608.616,Z 578.307,A -85,B 0,C 180,E1 -429.6,E2 -429.6} C_VEL
LIN {X 0,Y 608.567,Z 604.783,A -85,B 0,C 180,E1 -432.354,E2 -432.354} C_VEL
LIN {X 0,Y 608.511,Z 631.679,A -85,B 0,C 180,E1 -435.11,E2 -435.11} C_VEL
LIN {X 0,Y 608.497,Z 649.855,A -85,B 0,C 180,E1 -436.953,E2 -436.953} C_VEL
LIN {X 0,Y 608.531,Z 759.987,A -85,B 0,C 180,E1 -438.277,E2 -438.277} C_VEL
LIN {X 0,Y 608.535,Z 773.242,A -85,B 0,C 180,E1 -438.573,E2 -438.573} C_VEL
LIN {X 0,Y 608.543,Z 786.345,A -85,B 0,C 180,E1 -439.01,E2 -439.01} C_VEL
LIN {X 0,Y 608.501,Z 797.649,A -85,B 0,C 180,E1 -439.52,E2 -439.52} C_VEL
LIN {X 0,Y 608.474,Z 809.208,A -85,B 0,C 180,E1 -440.192,E2 -440.192} C_VEL
LIN {X 0,Y 608.485,Z 819.602,A -85,B 0,C 180,E1 -440.947,E2 -440.947} C_VEL
LIN {X 0,Y 608.475,Z 828.119,A -85,B 0,C 180,E1 -441.699,E2 -441.699} C_VEL
LIN {X 0,Y 608.47,Z 835.966,A -85,B 0,C 180,E1 -442.535,E2 -442.535} C_VEL
LIN {X 0,Y 608.46,Z 843.289,A -85,B 0,C 180,E1 -443.485,E2 -443.485} C_VEL
LIN {X 0,Y 608.45,Z 848.869,A -85,B 0,C 180,E1 -444.366,E2 -444.366} C_VEL
LIN {X 0,Y 608.432,Z 853.953,A -85,B 0,C 180,E1 -445.363,E2 -445.363} C_VEL
LIN {X 0,Y 608.449,Z 857.898,A -85,B 0,C 180,E1 -446.358,E2 -446.358} C_VEL
LIN {X 0,Y 608.425,Z 860.811,A -85,B 0,C 180,E1 -447.352,E2 -447.352} C_VEL
LIN {X 0,Y 608.441,Z 862.202,A -85,B 0,C 180,E1 -448.015,E2 -448.015} C_VEL
LIN {X 0,Y 608.438,Z 863.784,A -85,B 0,C 180,E1 -449.339,E2 -449.339} C_VEL
LIN {X 0,Y 608.434,Z 864,A -85,B 0,C 180,E1 -450.001,E2 -450.001} C_VEL
LIN {X 0,Y 608.448,Z 863.183,A -85,B 0,C 180,E1 -451.324,E2 -451.324} C_VEL
LIN {X 0,Y 608.441,Z 862.2,A -85,B 0,C 180,E1 -451.986,E2 -451.986} C_VEL
LIN {X 0,Y 608.425,Z 860.808,A -85,B 0,C 180,E1 -452.649,E2 -452.649} C_VEL
LIN {X 0,Y 608.449,Z 857.894,A -85,B 0,C 180,E1 -453.643,E2 -453.643} C_VEL
LIN {X 0,Y 608.432,Z 853.948,A -85,B 0,C 180,E1 -454.638,E2 -454.638} C_VEL
LIN {X 0,Y 608.437,Z 847.874,A -85,B 0,C 180,E1 -455.801,E2 -455.801} C_VEL
LIN {X 0,Y 608.462,Z 841.232,A -85,B 0,C 180,E1 -456.8,E2 -456.8} C_VEL
LIN {X 0,Y 608.456,Z 832.985,A -85,B 0,C 180,E1 -457.801,E2 -457.801} C_VEL
LIN {X 0,Y 608.472,Z 824.531,A -85,B 0,C 180,E1 -458.636,E2 -458.636} C_VEL
LIN {X 0,Y 608.471,Z 814.085,A -85,B 0,C 180,E1 -459.474,E2 -459.474} C_VEL
LIN {X 0,Y 608.487,Z 803.749,A -85,B 0,C 180,E1 -460.145,E2 -460.145} C_VEL
LIN {X 0,Y 608.521,Z 792.239,A -85,B 0,C 180,E1 -460.741,E2 -460.741} C_VEL
LIN {X 0,Y 608.538,Z 779.87,A -85,B 0,C 180,E1 -461.225,E2 -461.225} C_VEL
LIN {X 0,Y 608.534,Z 766.423,A -85,B 0,C 180,E1 -461.597,E2 -461.597} C_VEL
LIN {X 0,Y 608.539,Z 754.055,A -85,B 0,C 180,E1 -461.808,E2 -461.808} C_VEL
LIN {X 0,Y 608.512,Z 650.656,A -85,B 0,C 180,E1 -463.037,E2 -463.037} C_VEL
LIN {X 0,Y 608.527,Z 625.329,A -85,B 0,C 180,E1 -465.92,E2 -465.92} C_VEL
LIN {X 0,Y 608.563,Z 600.893,A -85,B 0,C 180,E1 -468.741,E2 -468.741} C_VEL
LIN {X 0,Y 608.602,Z 575.8,A -85,B 0,C 180,E1 -471.687,E2 -471.687} C_VEL
LIN {X 0,Y 608.672,Z 552.816,A -85,B 0,C 180,E1 -474.437,E2 -474.437} C_VEL
LIN {X 0,Y 608.712,Z 531.309,A -85,B 0,C 180,E1 -477.067,E2 -477.067} C_VEL
LIN {X 0,Y 608.739,Z 526.271,A -85,B 0,C 180,E1 -477.691,E2 -477.691} C_VEL
LIN {X 0,Y 608.467,Z 524.688,A -85,B 0,C 180,E1 -477.938,E2 -477.938} C_VEL
LIN {X 0,Y 608.471,Z 524.689,A -85,B 0,C 180,E1 -480.545,E2 -480.545} C_VEL
LIN {X 0,Y 608.461,Z 524.696,A -85,B 0,C 180,E1 -482.879,E2 -482.879} C_VEL
LIN {X 0,Y 608.452,Z 524.693,A -85,B 0,C 180,E1 -485.277,E2 -485.277} C_VEL
LIN {X 0,Y 608.466,Z 524.686,A -85,B 0,C 180,E1 -487.746,E2 -487.746} C_VEL
LIN {X 0,Y 608.447,Z 524.688,A -85,B 0,C 180,E1 -490.328,E2 -490.328} C_VEL
LIN {X 0,Y 608.48,Z 524.69,A -85,B 0,C 180,E1 -493.31,E2 -493.31} C_VEL
LIN {X 0,Y 608.47,Z 524.685,A -85,B 0,C 180,E1 -496.13,E2 -496.13} C_VEL
LIN {X 0,Y 608.459,Z 524.691,A -85,B 0,C 180,E1 -498.824,E2 -498.824} C_VEL
LIN {X 0,Y 608.475,Z 524.691,A -85,B 0,C 180,E1 -501.412,E2 -501.412} C_VEL
LIN {X 0,Y 608.477,Z 524.685,A -85,B 0,C 180,E1 -503.95,E2 -503.95} C_VEL
LIN {X 0,Y 608.448,Z 524.687,A -85,B 0,C 180,E1 -506.328,E2 -506.328} C_VEL
LIN {X 0,Y 608.46,Z 524.688,A -85,B 0,C 180,E1 -508.73,E2 -508.73} C_VEL
LIN {X 0,Y 608.475,Z 524.695,A -85,B 0,C 180,E1 -511.379,E2 -511.379} C_VEL
LIN {X 0,Y 608.468,Z 524.685,A -85,B 0,C 180,E1 -514.279,E2 -514.279} C_VEL
LIN {X 0,Y 608.451,Z 524.689,A -85,B 0,C 180,E1 -516.876,E2 -516.876} C_VEL
LIN {X 0,Y 608.468,Z 524.691,A -85,B 0,C 180,E1 -519.726,E2 -519.726} C_VEL
LIN {X 0,Y 608.448,Z 524.687,A -85,B 0,C 180,E1 -522.523,E2 -522.523} C_VEL
LIN {X 0,Y 608.479,Z 524.69,A -85,B 0,C 180,E1 -525.28,E2 -525.28} C_VEL
LIN {X 0,Y 608.465,Z 524.688,A -85,B 0,C 180,E1 -528,E2 -528} C_VEL
LIN {X 0,Y 608.462,Z 524.685,A -85,B 0,C 180,E1 -530.694,E2 -530.694} C_VEL
LIN {X 0,Y 608.476,Z 524.691,A -85,B 0,C 180,E1 -533.367,E2 -533.367} C_VEL
LIN {X 0,Y 608.455,Z 524.69,A -85,B 0,C 180,E1 -536.026,E2 -536.026} C_VEL
LIN {X 0,Y 608.468,Z 524.685,A -85,B 0,C 180,E1 -538.676,E2 -538.676} C_VEL
LIN {X 0,Y 608.468,Z 524.689,A -85,B 0,C 180,E1 -541.324,E2 -541.324} C_VEL
LIN {X 0,Y 608.458,Z 524.693,A -85,B 0,C 180,E1 -543.974,E2 -543.974} C_VEL
LIN {X 0,Y 608.476,Z 524.684,A -85,B 0,C 180,E1 -546.633,E2 -546.633} C_VEL
LIN {X 0,Y 608.456,Z 524.69,A -85,B 0,C 180,E1 -549.462,E2 -549.462} C_VEL
LIN {X 0,Y 607.785,Z 524.779,A -85,B 0,C 180,E1 -550.015,E2 -550.015} C_VEL
LIN {X 0,Y 604.935,Z 525.133,A -85,B 0,C 180,E1 -550.912,E2 -550.912} C_VEL
LIN {X 0,Y 602.529,Z 525.432,A -85,B 0,C 180,E1 -551.633,E2 -551.633} C_VEL
LIN {X 0,Y 601.495,Z 525.558,A -85,B 0,C 180,E1 -552.19,E2 -552.19} C_VEL
LIN {X 0,Y 601.411,Z 525.566,A -85,B 0,C 180,E1 -552.378,E2 -552.378} C_VEL
LIN {X 0,Y 601.425,Z 525.562,A -85,B 0,C 180,E1 -554.897,E2 -554.897} C_VEL
LIN {X 0,Y 601.43,Z 525.562,A -85,B 0,C 180,E1 -556.986,E2 -556.986} C_VEL
LIN {X 0,Y 601.404,Z 525.573,A -85,B 0,C 180,E1 -559.81,E2 -559.81} C_VEL
LIN {X 0,Y 601.411,Z 525.565,A -85,B 0,C 180,E1 -562.683,E2 -562.683} C_VEL
LIN {X 0,Y 601.402,Z 525.565,A -85,B 0,C 180,E1 -564.879,E2 -564.879} C_VEL
LIN {X 0,Y 601.419,Z 525.571,A -85,B 0,C 180,E1 -567.868,E2 -567.868} C_VEL
LIN {X 0,Y 601.429,Z 525.571,A -85,B 0,C 180,E1 -570.164,E2 -570.164} C_VEL
LIN {X 0,Y 601.418,Z 525.565,A -85,B 0,C 180,E1 -572.715,E2 -572.715} C_VEL
LIN {X 0,Y 601.391,Z 525.566,A -85,B 0,C 180,E1 -575.112,E2 -575.112} C_VEL
LIN {X 0,Y 601.437,Z 525.562,A -85,B 0,C 180,E1 -577.419,E2 -577.419} C_VEL
LIN {X 0,Y 601.411,Z 525.572,A -85,B 0,C 180,E1 -579.995,E2 -579.995} C_VEL
LIN {X 0,Y 601.413,Z 525.567,A -85,B 0,C 180,E1 -582.67,E2 -582.67} C_VEL
LIN {X 0,Y 601.426,Z 525.568,A -85,B 0,C 180,E1 -584.535,E2 -584.535} C_VEL
LIN {X 0,Y 601.409,Z 525.563,A -85,B 0,C 180,E1 -587.41,E2 -587.41} C_VEL
LIN {X 0,Y 601.404,Z 525.57,A -85,B 0,C 180,E1 -590.004,E2 -590.004} C_VEL
LIN {X 0,Y 601.435,Z 525.567,A -85,B 0,C 180,E1 -592.618,E2 -592.618} C_VEL
LIN {X 0,Y 601.433,Z 525.562,A -85,B 0,C 180,E1 -595.069,E2 -595.069} C_VEL
LIN {X 0,Y 601.434,Z 525.561,A -85,B 0,C 180,E1 -597.484,E2 -597.484} C_VEL
LIN {X 0,Y 601.431,Z 525.564,A -85,B 0,C 180,E1 -599.852,E2 -599.852} C_VEL
LIN {X 0,Y 601.414,Z 525.573,A -85,B 0,C 180,E1 -602.639,E2 -602.639} C_VEL
LIN {X 0,Y 601.437,Z 525.738,A -85,B 0,C 180,E1 -605.393,E2 -605.393} C_VEL
LIN {X 0,Y 601.815,Z 527.49,A -85,B 0,C 180,E1 -605.629,E2 -605.629} C_VEL
LIN {X 0,Y 601.721,Z 548.567,A -85,B 0,C 180,E1 -608.233,E2 -608.233} C_VEL
LIN {X 0,Y 601.63,Z 572.398,A -85,B 0,C 180,E1 -611.123,E2 -611.123} C_VEL
LIN {X 0,Y 601.546,Z 597.069,A -85,B 0,C 180,E1 -614.064,E2 -614.064} C_VEL
LIN {X 0,Y 601.503,Z 621.048,A -85,B 0,C 180,E1 -616.862,E2 -616.862} C_VEL
LIN {X 0,Y 601.609,Z 729.791,A -85,B 0,C 180,E1 -618.182,E2 -618.182} C_VEL
LIN {X 0,Y 601.592,Z 743.133,A -85,B 0,C 180,E1 -618.48,E2 -618.48} C_VEL
LIN {X 0,Y 601.539,Z 755.563,A -85,B 0,C 180,E1 -618.895,E2 -618.895} C_VEL
LIN {X 0,Y 601.537,Z 766.742,A -85,B 0,C 180,E1 -619.396,E2 -619.396} C_VEL
LIN {X 0,Y 601.479,Z 778.519,A -85,B 0,C 180,E1 -620.075,E2 -620.075} C_VEL
LIN {X 0,Y 601.444,Z 789.029,A -85,B 0,C 180,E1 -620.838,E2 -620.838} C_VEL
LIN {X 0,Y 601.429,Z 797.638,A -85,B 0,C 180,E1 -621.6,E2 -621.6} C_VEL
LIN {X 0,Y 601.418,Z 805.567,A -85,B 0,C 180,E1 -622.445,E2 -622.445} C_VEL
LIN {X 0,Y 601.377,Z 812.886,A -85,B 0,C 180,E1 -623.393,E2 -623.393} C_VEL
LIN {X 0,Y 601.372,Z 818.608,A -85,B 0,C 180,E1 -624.299,E2 -624.299} C_VEL
LIN {X 0,Y 601.335,Z 823.751,A -85,B 0,C 180,E1 -625.307,E2 -625.307} C_VEL
LIN {X 0,Y 601.367,Z 827.74,A -85,B 0,C 180,E1 -626.314,E2 -626.314} C_VEL
LIN {X 0,Y 601.324,Z 830.69,A -85,B 0,C 180,E1 -627.32,E2 -627.32} C_VEL
LIN {X 0,Y 601.341,Z 832.126,A -85,B 0,C 180,E1 -627.99,E2 -627.99} C_VEL
LIN {X 0,Y 601.339,Z 833.752,A -85,B 0,C 180,E1 -629.33,E2 -629.33} C_VEL
LIN {X 0,Y 601.336,Z 833.995,A -85,B 0,C 180,E1 -629.999,E2 -629.999} C_VEL
LIN {X 0,Y 601.339,Z 833.815,A -85,B 0,C 180,E1 -630.669,E2 -630.669} C_VEL
LIN {X 0,Y 601.342,Z 832.276,A -85,B 0,C 180,E1 -632.009,E2 -632.009} C_VEL
LIN {X 0,Y 601.326,Z 830.918,A -85,B 0,C 180,E1 -632.679,E2 -632.679} C_VEL
LIN {X 0,Y 601.368,Z 828.043,A -85,B 0,C 180,E1 -633.685,E2 -633.685} C_VEL
LIN {X 0,Y 601.337,Z 824.145,A -85,B 0,C 180,E1 -634.692,E2 -634.692} C_VEL
LIN {X 0,Y 601.373,Z 819.115,A -85,B 0,C 180,E1 -635.7,E2 -635.7} C_VEL
LIN {X 0,Y 601.382,Z 812.795,A -85,B 0,C 180,E1 -636.71,E2 -636.71} C_VEL
LIN {X 0,Y 601.396,Z 804.883,A -85,B 0,C 180,E1 -637.723,E2 -637.723} C_VEL
LIN {X 0,Y 601.436,Z 795.037,A -85,B 0,C 180,E1 -638.737,E2 -638.737} C_VEL
LIN {X 0,Y 601.447,Z 784.719,A -85,B 0,C 180,E1 -639.584,E2 -639.584} C_VEL
LIN {X 0,Y 601.494,Z 773.108,A -85,B 0,C 180,E1 -640.348,E2 -640.348} C_VEL
LIN {X 0,Y 601.553,Z 760.812,A -85,B 0,C 180,E1 -640.975,E2 -640.975} C_VEL
LIN {X 0,Y 601.57,Z 748.277,A -85,B 0,C 180,E1 -641.455,E2 -641.455} C_VEL
LIN {X 0,Y 601.599,Z 735.662,A -85,B 0,C 180,E1 -641.796,E2 -641.796} C_VEL
LIN {X 0,Y 601.61,Z 722.56,A -85,B 0,C 180,E1 -642.009,E2 -642.009} C_VEL
LIN {X 0,Y 601.542,Z 622.376,A -85,B 0,C 180,E1 -643.211,E2 -643.211} C_VEL
LIN {X 0,Y 601.474,Z 621.379,A -85,B 0,C 180,E1 -643.256,E2 -643.256} C_VEL
LIN {X 0,Y 601.528,Z 598.404,A -85,B 0,C 180,E1 -646.284,E2 -646.284} C_VEL
LIN {X 0,Y 601.583,Z 577.396,A -85,B 0,C 180,E1 -649.093,E2 -649.093} C_VEL
LIN {X 0,Y 601.67,Z 556.388,A -85,B 0,C 180,E1 -651.948,E2 -651.948} C_VEL
LIN {X 0,Y 601.759,Z 536.491,A -85,B 0,C 180,E1 -654.706,E2 -654.706} C_VEL
LIN {X 0,Y 601.666,Z 526.755,A -85,B 0,C 180,E1 -656.083,E2 -656.083} C_VEL
LIN {X 0,Y 601.417,Z 525.569,A -85,B 0,C 180,E1 -656.295,E2 -656.295} C_VEL
LIN {X 0,Y 601.441,Z 525.565,A -85,B 0,C 180,E1 -658.789,E2 -658.789} C_VEL
LIN {X 0,Y 601.413,Z 525.567,A -85,B 0,C 180,E1 -661.725,E2 -661.725} C_VEL
LIN {X 0,Y 601.43,Z 525.562,A -85,B 0,C 180,E1 -664.117,E2 -664.117} C_VEL
LIN {X 0,Y 601.413,Z 525.565,A -85,B 0,C 180,E1 -666.581,E2 -666.581} C_VEL
LIN {X 0,Y 601.44,Z 525.567,A -85,B 0,C 180,E1 -669.535,E2 -669.535} C_VEL
LIN {X 0,Y 601.422,Z 525.566,A -85,B 0,C 180,E1 -671.764,E2 -671.764} C_VEL
LIN {X 0,Y 601.418,Z 525.563,A -85,B 0,C 180,E1 -674.534,E2 -674.534} C_VEL
LIN {X 0,Y 601.435,Z 525.572,A -85,B 0,C 180,E1 -677.405,E2 -677.405} C_VEL
LIN {X 0,Y 601.436,Z 525.561,A -85,B 0,C 180,E1 -680.463,E2 -680.463} C_VEL
LIN {X 0,Y 601.413,Z 525.575,A -85,B 0,C 180,E1 -683.418,E2 -683.418} C_VEL
LIN {X 0,Y 601.474,Z 525.745,A -85,B 0,C 180,E1 -685.158,E2 -685.158} C_VEL
LIN {X 0,Y 601.627,Z 595.488,A -85,B 0,C 180,E1 -685.996,E2 -685.996} C_VEL
LIN {X 0,Y 601.571,Z 613.158,A -85,B 0,C 180,E1 -686.244,E2 -686.244} C_VEL
LIN {X 0,Y 601.556,Z 625.421,A -85,B 0,C 180,E1 -686.544,E2 -686.544} C_VEL
LIN {X 0,Y 601.553,Z 638.225,A -85,B 0,C 180,E1 -687.005,E2 -687.005} C_VEL
LIN {X 0,Y 601.496,Z 650.318,A -85,B 0,C 180,E1 -687.587,E2 -687.587} C_VEL
LIN {X 0,Y 601.468,Z 661.538,A -85,B 0,C 180,E1 -688.277,E2 -688.277} C_VEL
LIN {X 0,Y 601.43,Z 671.691,A -85,B 0,C 180,E1 -689.058,E2 -689.058} C_VEL
LIN {X 0,Y 601.399,Z 680.165,A -85,B 0,C 180,E1 -689.854,E2 -689.854} C_VEL
LIN {X 0,Y 601.37,Z 688.241,A -85,B 0,C 180,E1 -690.772,E2 -690.772} C_VEL
LIN {X 0,Y 601.374,Z 695.264,A -85,B 0,C 180,E1 -691.751,E2 -691.751} C_VEL
LIN {X 0,Y 601.341,Z 701.731,A -85,B 0,C 180,E1 -692.883,E2 -692.883} C_VEL
LIN {X 0,Y 601.336,Z 707.125,A -85,B 0,C 180,E1 -694.145,E2 -694.145} C_VEL
LIN {X 0,Y 601.338,Z 710.162,A -85,B 0,C 180,E1 -695.118,E2 -695.118} C_VEL
LIN {X 0,Y 601.347,Z 711.866,A -85,B 0,C 180,E1 -695.855,E2 -695.855} C_VEL
LIN {X 0,Y 601.324,Z 713.043,A -85,B 0,C 180,E1 -696.586,E2 -696.586} C_VEL
LIN {X 0,Y 601.339,Z 713.808,A -85,B 0,C 180,E1 -697.409,E2 -697.409} C_VEL
LIN {X 0,Y 601.332,Z 714,A -85,B 0,C 180,E1 -698.038,E2 -698.038} C_VEL
LIN {X 0,Y 601.337,Z 713.372,A -85,B 0,C 180,E1 -699.221,E2 -699.221} C_VEL
LIN {X 0,Y 601.315,Z 711.968,A -85,B 0,C 180,E1 -700.187,E2 -700.187} C_VEL
LIN {X 0,Y 601.341,Z 709.56,A -85,B 0,C 180,E1 -701.198,E2 -701.198} C_VEL
LIN {X 0,Y 601.345,Z 705.749,A -85,B 0,C 180,E1 -702.31,E2 -702.31} C_VEL
LIN {X 0,Y 601.36,Z 700.754,A -85,B 0,C 180,E1 -703.395,E2 -703.395} C_VEL
LIN {X 0,Y 601.355,Z 694.818,A -85,B 0,C 180,E1 -704.407,E2 -704.407} C_VEL
LIN {X 0,Y 601.398,Z 687.188,A -85,B 0,C 180,E1 -705.448,E2 -705.448} C_VEL
LIN {X 0,Y 601.421,Z 679.109,A -85,B 0,C 180,E1 -706.346,E2 -706.346} C_VEL
LIN {X 0,Y 601.461,Z 668.933,A -85,B 0,C 180,E1 -707.258,E2 -707.258} C_VEL
LIN {X 0,Y 601.468,Z 658.278,A -85,B 0,C 180,E1 -708.03,E2 -708.03} C_VEL
LIN {X 0,Y 601.512,Z 646.686,A -85,B 0,C 180,E1 -708.697,E2 -708.697} C_VEL
LIN {X 0,Y 601.559,Z 633.613,A -85,B 0,C 180,E1 -709.269,E2 -709.269} C_VEL
LIN {X 0,Y 601.579,Z 620.784,A -85,B 0,C 180,E1 -709.674,E2 -709.674} C_VEL
LIN {X 0,Y 601.584,Z 608.464,A -85,B 0,C 180,E1 -709.929,E2 -709.929} C_VEL
LIN {X 0,Y 601.546,Z 526.2,A -85,B 0,C 180,E1 -710.925,E2 -710.925} C_VEL
LIN {X 0,Y 601.436,Z 525.567,A -85,B 0,C 180,E1 -710.966,E2 -710.966} C_VEL
LIN {X 0,Y 601.444,Z 525.562,A -85,B 0,C 180,E1 -713.323,E2 -713.323} C_VEL
LIN {X 0,Y 601.402,Z 525.567,A -85,B 0,C 180,E1 -715.979,E2 -715.979} C_VEL
LIN {X 0,Y 601.431,Z 525.573,A -85,B 0,C 180,E1 -718.661,E2 -718.661} C_VEL
LIN {X 0,Y 601.423,Z 525.564,A -85,B 0,C 180,E1 -721.339,E2 -721.339} C_VEL
LIN {X 0,Y 601.428,Z 525.564,A -85,B 0,C 180,E1 -723.35,E2 -723.35} C_VEL
LIN {X 0,Y 601.426,Z 525.564,A -85,B 0,C 180,E1 -726.037,E2 -726.037} C_VEL
LIN {X 0,Y 601.435,Z 525.572,A -85,B 0,C 180,E1 -728.738,E2 -728.738} C_VEL
LIN {X 0,Y 601.427,Z 525.563,A -85,B 0,C 180,E1 -731.458,E2 -731.458} C_VEL
LIN {X 0,Y 601.408,Z 525.567,A -85,B 0,C 180,E1 -734.206,E2 -734.206} C_VEL
LIN {X 0,Y 601.425,Z 525.569,A -85,B 0,C 180,E1 -736.986,E2 -736.986} C_VEL
LIN {X 0,Y 601.401,Z 525.565,A -85,B 0,C 180,E1 -739.81,E2 -739.81} C_VEL
LIN {X 0,Y 601.406,Z 525.573,A -85,B 0,C 180,E1 -742.607,E2 -742.607} C_VEL
LIN {X 0,Y 601.4,Z 525.575,A -85,B 0,C 180,E1 -744.879,E2 -744.879} C_VEL
LIN {X 0,Y 601.417,Z 525.563,A -85,B 0,C 180,E1 -747.868,E2 -747.868} C_VEL
LIN {X 0,Y 601.44,Z 525.562,A -85,B 0,C 180,E1 -750.163,E2 -750.163} C_VEL
LIN {X 0,Y 601.42,Z 525.573,A -85,B 0,C 180,E1 -752.717,E2 -752.717} C_VEL
LIN {X 0,Y 601.414,Z 525.569,A -85,B 0,C 180,E1 -755.117,E2 -755.117} C_VEL
LIN {X 0,Y 601.431,Z 525.563,A -85,B 0,C 180,E1 -757.419,E2 -757.419} C_VEL
LIN {X 0,Y 601.412,Z 525.564,A -85,B 0,C 180,E1 -759.995,E2 -759.995} C_VEL
LIN {X 0,Y 601.435,Z 525.569,A -85,B 0,C 180,E1 -762.668,E2 -762.668} C_VEL
LIN {X 0,Y 601.419,Z 525.565,A -85,B 0,C 180,E1 -765.483,E2 -765.483} C_VEL
LIN {X 0,Y 601.424,Z 525.566,A -85,B 0,C 180,E1 -768.407,E2 -768.407} C_VEL
LIN {X 0,Y 601.439,Z 525.572,A -85,B 0,C 180,E1 -770.877,E2 -770.877} C_VEL
LIN {X 0,Y 601.441,Z 525.561,A -85,B 0,C 180,E1 -773.735,E2 -773.735} C_VEL
LIN {X 0,Y 601.429,Z 525.57,A -85,B 0,C 180,E1 -776.688,E2 -776.688} C_VEL
LIN {X 0,Y 601.427,Z 525.571,A -85,B 0,C 180,E1 -779.06,E2 -779.06} C_VEL
LIN {X 0,Y 601.434,Z 525.566,A -85,B 0,C 180,E1 -781.374,E2 -781.374} C_VEL
LIN {X 0,Y 601.449,Z 525.672,A -85,B 0,C 180,E1 -783.628,E2 -783.628} C_VEL
LIN {X 0,Y 601.966,Z 529.034,A -85,B 0,C 180,E1 -784.025,E2 -784.025} C_VEL
LIN {X 0,Y 601.84,Z 554.522,A -85,B 0,C 180,E1 -786.808,E2 -786.808} C_VEL
LIN {X 0,Y 601.743,Z 579.569,A -85,B 0,C 180,E1 -789.49,E2 -789.49} C_VEL
LIN {X 0,Y 601.631,Z 606.464,A -85,B 0,C 180,E1 -792.32,E2 -792.32} C_VEL
LIN {X 0,Y 601.534,Z 633.36,A -85,B 0,C 180,E1 -795.107,E2 -795.107} C_VEL
LIN {X 0,Y 601.521,Z 649.75,A -85,B 0,C 180,E1 -796.788,E2 -796.788} C_VEL
LIN {X 0,Y 601.672,Z 661.151,A -85,B 0,C 180,E1 -796.942,E2 -796.942} C_VEL
LIN {X 0,Y 601.598,Z 759.987,A -85,B 0,C 180,E1 -798.14,E2 -798.14} C_VEL
LIN {X 0,Y 601.579,Z 773.242,A -85,B 0,C 180,E1 -798.439,E2 -798.439} C_VEL
LIN {X 0,Y 601.548,Z 784.938,A -85,B 0,C 180,E1 -798.827,E2 -798.827} C_VEL
LIN {X 0,Y 601.515,Z 795.938,A -85,B 0,C 180,E1 -799.312,E2 -799.312} C_VEL
LIN {X 0,Y 601.47,Z 806.592,A -85,B 0,C 180,E1 -799.906,E2 -799.906} C_VEL
LIN {X 0,Y 601.445,Z 817.484,A -85,B 0,C 180,E1 -800.67,E2 -800.67} C_VEL
LIN {X 0,Y 601.429,Z 828.119,A -85,B 0,C 180,E1 -801.602,E2 -801.602} C_VEL
LIN {X 0,Y 601.417,Z 835.966,A -85,B 0,C 180,E1 -802.446,E2 -802.446} C_VEL
LIN {X 0,Y 601.369,Z 843.228,A -85,B 0,C 180,E1 -803.398,E2 -803.398} C_VEL
LIN {X 0,Y 601.371,Z 848.87,A -85,B 0,C 180,E1 -804.3,E2 -804.3} C_VEL
LIN {X 0,Y 601.336,Z 853.953,A -85,B 0,C 180,E1 -805.308,E2 -805.308} C_VEL
LIN {X 0,Y 601.368,Z 857.898,A -85,B 0,C 180,E1 -806.315,E2 -806.315} C_VEL
LIN {X 0,Y 601.325,Z 860.811,A -85,B 0,C 180,E1 -807.321,E2 -807.321} C_VEL
LIN {X 0,Y 601.34,Z 862.203,A -85,B 0,C 180,E1 -807.991,E2 -807.991} C_VEL
LIN {X 0,Y 601.339,Z 863.784,A -85,B 0,C 180,E1 -809.331,E2 -809.331} C_VEL
LIN {X 0,Y 601.335,Z 864,A -85,B 0,C 180,E1 -810.001,E2 -810.001} C_VEL
LIN {X 0,Y 601.348,Z 863.183,A -85,B 0,C 180,E1 -811.34,E2 -811.34} C_VEL
LIN {X 0,Y 601.34,Z 862.201,A -85,B 0,C 180,E1 -812.01,E2 -812.01} C_VEL
LIN {X 0,Y 601.325,Z 860.808,A -85,B 0,C 180,E1 -812.68,E2 -812.68} C_VEL
LIN {X 0,Y 601.368,Z 857.894,A -85,B 0,C 180,E1 -813.686,E2 -813.686} C_VEL
LIN {X 0,Y 601.336,Z 853.948,A -85,B 0,C 180,E1 -814.693,E2 -814.693} C_VEL
LIN {X 0,Y 601.372,Z 847.874,A -85,B 0,C 180,E1 -815.87,E2 -815.87} C_VEL
LIN {X 0,Y 601.382,Z 841.232,A -85,B 0,C 180,E1 -816.88,E2 -816.88} C_VEL
LIN {X 0,Y 601.4,Z 832.985,A -85,B 0,C 180,E1 -817.893,E2 -817.893} C_VEL
LIN {X 0,Y 601.436,Z 824.532,A -85,B 0,C 180,E1 -818.738,E2 -818.738} C_VEL
LIN {X 0,Y 601.44,Z 814.086,A -85,B 0,C 180,E1 -819.586,E2 -819.586} C_VEL
LIN {X 0,Y 601.489,Z 803.75,A -85,B 0,C 180,E1 -820.265,E2 -820.265} C_VEL
LIN {X 0,Y 601.537,Z 792.896,A -85,B 0,C 180,E1 -820.836,E2 -820.836} C_VEL
LIN {X 0,Y 601.567,Z 780.368,A -85,B 0,C 180,E1 -821.341,E2 -821.341} C_VEL
LIN {X 0,Y 601.594,Z 767.337,A -85,B 0,C 180,E1 -821.712,E2 -821.712} C_VEL
LIN {X 0,Y 601.606,Z 754.055,A -85,B 0,C 180,E1 -821.946,E2 -821.946} C_VEL
LIN {X 0,Y 601.574,Z 651.33,A -85,B 0,C 180,E1 -823.178,E2 -823.178} C_VEL
LIN {X 0,Y 601.477,Z 650.468,A -85,B 0,C 180,E1 -823.214,E2 -823.214} C_VEL
LIN {X 0,Y 601.545,Z 626.829,A -85,B 0,C 180,E1 -825.936,E2 -825.936} C_VEL
LIN {X 0,Y 601.62,Z 603.727,A -85,B 0,C 180,E1 -828.631,E2 -828.631} C_VEL
LIN {X 0,Y 601.723,Z 580.302,A -85,B 0,C 180,E1 -831.407,E2 -831.407} C_VEL
LIN {X 0,Y 601.819,Z 556.779,A -85,B 0,C 180,E1 -834.248,E2 -834.248} C_VEL
LIN {X 0,Y 601.957,Z 533.775,A -85,B 0,C 180,E1 -837.087,E2 -837.087} C_VEL
LIN {X 0,Y 601.889,Z 527.772,A -85,B 0,C 180,E1 -837.844,E2 -837.844} C_VEL
LIN {X 0,Y 601.416,Z 525.569,A -85,B 0,C 180,E1 -838.152,E2 -838.152} C_VEL
LIN {X 0,Y 601.433,Z 525.573,A -85,B 0,C 180,E1 -840.941,E2 -840.941} C_VEL
LIN {X 0,Y 601.43,Z 525.567,A -85,B 0,C 180,E1 -843.313,E2 -843.313} C_VEL
LIN {X 0,Y 601.392,Z 525.567,A -85,B 0,C 180,E1 -845.754,E2 -845.754} C_VEL
LIN {X 0,Y 601.433,Z 525.563,A -85,B 0,C 180,E1 -848.471,E2 -848.471} C_VEL
LIN {X 0,Y 601.418,Z 525.571,A -85,B 0,C 180,E1 -850.874,E2 -850.874} C_VEL
LIN {X 0,Y 601.431,Z 525.564,A -85,B 0,C 180,E1 -853.586,E2 -853.586} C_VEL
LIN {X 0,Y 601.451,Z 525.56,A -85,B 0,C 180,E1 -856.425,E2 -856.425} C_VEL
LIN {X 0,Y 601.421,Z 525.569,A -85,B 0,C 180,E1 -859.426,E2 -859.426} C_VEL
LIN {X 0,Y 601.425,Z 525.565,A -85,B 0,C 180,E1 -861.732,E2 -861.732} C_VEL
LIN {X 0,Y 601.406,Z 525.564,A -85,B 0,C 180,E1 -864.246,E2 -864.246} C_VEL
LIN {X 0,Y 601.418,Z 525.565,A -85,B 0,C 180,E1 -866.686,E2 -866.686} C_VEL
LIN {X 0,Y 601.424,Z 525.569,A -85,B 0,C 180,E1 -869.058,E2 -869.058} C_VEL
LIN {X 0,Y 601.435,Z 525.572,A -85,B 0,C 180,E1 -871.373,E2 -871.373} C_VEL
LIN {X 0,Y 601.403,Z 525.57,A -85,B 0,C 180,E1 -873.636,E2 -873.636} C_VEL
LIN {X 0,Y 601.42,Z 525.563,A -85,B 0,C 180,E1 -876.59,E2 -876.59} C_VEL
LIN {X 0,Y 601.437,Z 525.571,A -85,B 0,C 180,E1 -879.478,E2 -879.478} C_VEL
LIN {X 0,Y 601.396,Z 525.565,A -85,B 0,C 180,E1 -882.312,E2 -882.312} C_VEL
LIN {X 0,Y 601.411,Z 525.564,A -85,B 0,C 180,E1 -884.409,E2 -884.409} C_VEL
LIN {X 0,Y 601.422,Z 525.567,A -85,B 0,C 180,E1 -887.172,E2 -887.172} C_VEL
LIN {X 0,Y 601.438,Z 525.565,A -85,B 0,C 180,E1 -889.905,E2 -889.905} C_VEL
LIN {X 0,Y 601.437,Z 525.561,A -85,B 0,C 180,E1 -892.615,E2 -892.615} C_VEL
LIN {X 0,Y 601.432,Z 525.567,A -85,B 0,C 180,E1 -895.308,E2 -895.308} C_VEL
LIN {X 0,Y 601.425,Z 525.567,A -85,B 0,C 180,E1 -897.991,E2 -897.991} C_VEL
LIN {X 0,Y 601.45,Z 525.559,A -85,B 0,C 180,E1 -900.67,E2 -900.67} C_VEL
LIN {X 0,Y 601.426,Z 525.566,A -85,B 0,C 180,E1 -903.35,E2 -903.35} C_VEL
LIN {X 0,Y 601.417,Z 525.569,A -85,B 0,C 180,E1 -906.037,E2 -906.037} C_VEL
LIN {X 0,Y 601.437,Z 525.561,A -85,B 0,C 180,E1 -908.738,E2 -908.738} C_VEL
LIN {X 0,Y 601.432,Z 525.566,A -85,B 0,C 180,E1 -911.458,E2 -911.458} C_VEL
LIN {X 0,Y 601.411,Z 525.566,A -85,B 0,C 180,E1 -912.378,E2 -912.378} C_VEL
LIN {X 0,Y 600.743,Z 525.649,A -85,B 0,C 180,E1 -912.938,E2 -912.938} C_VEL
LIN {X 0,Y 597.89,Z 526.013,A -85,B 0,C 180,E1 -913.846,E2 -913.846} C_VEL
LIN {X 0,Y 595.48,Z 526.307,A -85,B 0,C 180,E1 -914.576,E2 -914.576} C_VEL
LIN {X 0,Y 594.444,Z 526.433,A -85,B 0,C 180,E1 -915.139,E2 -915.139} C_VEL
LIN {X 0,Y 594.358,Z 526.445,A -85,B 0,C 180,E1 -915.33,E2 -915.33} C_VEL
LIN {X 0,Y 594.38,Z 526.451,A -85,B 0,C 180,E1 -917.904,E2 -917.904} C_VEL
LIN {X 0,Y 594.379,Z 526.44,A -85,B 0,C 180,E1 -920.917,E2 -920.917} C_VEL
LIN {X 0,Y 594.391,Z 526.444,A -85,B 0,C 180,E1 -923.704,E2 -923.704} C_VEL
LIN {X 0,Y 594.383,Z 526.44,A -85,B 0,C 180,E1 -926.7,E2 -926.7} C_VEL
LIN {X 0,Y 594.38,Z 526.44,A -85,B 0,C 180,E1 -928.999,E2 -928.999} C_VEL
LIN {X 0,Y 594.377,Z 526.443,A -85,B 0,C 180,E1 -931.643,E2 -931.643} C_VEL
LIN {X 0,Y 594.378,Z 526.443,A -85,B 0,C 180,E1 -934.58,E2 -934.58} C_VEL
LIN {X 0,Y 594.392,Z 526.441,A -85,B 0,C 180,E1 -937.609,E2 -937.609} C_VEL
LIN {X 0,Y 594.371,Z 526.446,A -85,B 0,C 180,E1 -940.567,E2 -940.567} C_VEL
LIN {X 0,Y 594.382,Z 526.439,A -85,B 0,C 180,E1 -943.298,E2 -943.298} C_VEL
LIN {X 0,Y 594.362,Z 526.452,A -85,B 0,C 180,E1 -946.161,E2 -946.161} C_VEL
LIN {X 0,Y 594.378,Z 526.447,A -85,B 0,C 180,E1 -948.536,E2 -948.536} C_VEL
LIN {X 0,Y 594.375,Z 526.44,A -85,B 0,C 180,E1 -951.297,E2 -951.297} C_VEL
LIN {X 0,Y 594.354,Z 526.445,A -85,B 0,C 180,E1 -953.756,E2 -953.756} C_VEL
LIN {X 0,Y 594.382,Z 526.448,A -85,B 0,C 180,E1 -956.239,E2 -956.239} C_VEL
LIN {X 0,Y 594.371,Z 526.449,A -85,B 0,C 180,E1 -958.65,E2 -958.65} C_VEL
LIN {X 0,Y 594.387,Z 526.442,A -85,B 0,C 180,E1 -961.042,E2 -961.042} C_VEL
LIN {X 0,Y 594.39,Z 526.443,A -85,B 0,C 180,E1 -963.977,E2 -963.977} C_VEL
LIN {X 0,Y 594.393,Z 526.531,A -85,B 0,C 180,E1 -965.182,E2 -965.182} C_VEL
LIN {X 0,Y 594.966,Z 529.466,A -85,B 0,C 180,E1 -965.579,E2 -965.579} C_VEL
LIN {X 0,Y 594.827,Z 550.042,A -85,B 0,C 180,E1 -968.15,E2 -968.15} C_VEL
LIN {X 0,Y 594.695,Z 574.155,A -85,B 0,C 180,E1 -971.108,E2 -971.108} C_VEL
LIN {X 0,Y 594.584,Z 598.544,A -85,B 0,C 180,E1 -974.049,E2 -974.049} C_VEL
LIN {X 0,Y 594.508,Z 621.094,A -85,B 0,C 180,E1 -976.705,E2 -976.705} C_VEL
LIN {X 0,Y 594.754,Z 636.294,A -85,B 0,C 180,E1 -976.895,E2 -976.895} C_VEL
LIN {X 0,Y 594.662,Z 729.812,A -85,B 0,C 180,E1 -978.042,E2 -978.042} C_VEL
LIN {X 0,Y 594.626,Z 743.159,A -85,B 0,C 180,E1 -978.344,E2 -978.344} C_VEL
LIN {X 0,Y 594.554,Z 756.407,A -85,B 0,C 180,E1 -978.795,E2 -978.795} C_VEL
LIN {X 0,Y 594.517,Z 768.391,A -85,B 0,C 180,E1 -979.355,E2 -979.355} C_VEL
LIN {X 0,Y 594.468,Z 779.807,A -85,B 0,C 180,E1 -980.043,E2 -980.043} C_VEL
LIN {X 0,Y 594.406,Z 790.094,A -85,B 0,C 180,E1 -980.815,E2 -980.815} C_VEL
LIN {X 0,Y 594.373,Z 799.362,A -85,B 0,C 180,E1 -981.671,E2 -981.671} C_VEL
LIN {X 0,Y 594.317,Z 808.333,A -85,B 0,C 180,E1 -982.696,E2 -982.696} C_VEL
LIN {X 0,Y 594.285,Z 814.856,A -85,B 0,C 180,E1 -983.612,E2 -983.612} C_VEL
LIN {X 0,Y 594.289,Z 820.441,A -85,B 0,C 180,E1 -984.571,E2 -984.571} C_VEL
LIN {X 0,Y 594.27,Z 825.183,A -85,B 0,C 180,E1 -985.591,E2 -985.591} C_VEL
LIN {X 0,Y 594.267,Z 828.815,A -85,B 0,C 180,E1 -986.61,E2 -986.61} C_VEL
LIN {X 0,Y 594.225,Z 830.691,A -85,B 0,C 180,E1 -987.288,E2 -987.288} C_VEL
LIN {X 0,Y 594.24,Z 832.127,A -85,B 0,C 180,E1 -987.966,E2 -987.966} C_VEL
LIN {X 0,Y 594.24,Z 833.752,A -85,B 0,C 180,E1 -989.322,E2 -989.322} C_VEL
LIN {X 0,Y 594.236,Z 833.996,A -85,B 0,C 180,E1 -989.999,E2 -989.999} C_VEL
LIN {X 0,Y 594.239,Z 833.815,A -85,B 0,C 180,E1 -990.677,E2 -990.677} C_VEL
LIN {X 0,Y 594.241,Z 832.275,A -85,B 0,C 180,E1 -992.033,E2 -992.033} C_VEL
LIN {X 0,Y 594.226,Z 830.917,A -85,B 0,C 180,E1 -992.711,E2 -992.711} C_VEL
LIN {X 0,Y 594.289,Z 828.042,A -85,B 0,C 180,E1 -993.729,E2 -993.729} C_VEL
LIN {X 0,Y 594.242,Z 824.144,A -85,B 0,C 180,E1 -994.748,E2 -994.748} C_VEL
LIN {X 0,Y 594.299,Z 819.114,A -85,B 0,C 180,E1 -995.768,E2 -995.768} C_VEL
LIN {X 0,Y 594.316,Z 812.789,A -85,B 0,C 180,E1 -996.791,E2 -996.791} C_VEL
LIN {X 0,Y 594.346,Z 804.88,A -85,B 0,C 180,E1 -997.815,E2 -997.815} C_VEL
LIN {X 0,Y 594.381,Z 795.03,A -85,B 0,C 180,E1 -998.841,E2 -998.841} C_VEL
LIN {X 0,Y 594.429,Z 784.714,A -85,B 0,C 180,E1 -999.699,E2 -999.699} C_VEL
LIN {X 0,Y 594.509,Z 773.103,A -85,B 0,C 180,E1 -1000.471,E2 -1000.471} C_VEL
LIN {X 0,Y 594.571,Z 761.167,A -85,B 0,C 180,E1 -1001.089,E2 -1001.089} C_VEL
LIN {X 0,Y 594.62,Z 748.266,A -85,B 0,C 180,E1 -1001.59,E2 -1001.59} C_VEL
LIN {X 0,Y 594.666,Z 735.63,A -85,B 0,C 180,E1 -1001.935,E2 -1001.935} C_VEL
LIN {X 0,Y 594.681,Z 722.515,A -85,B 0,C 180,E1 -1002.151,E2 -1002.151} C_VEL
LIN {X 0,Y 594.657,Z 623.224,A -85,B 0,C 180,E1 -1003.356,E2 -1003.356} C_VEL
LIN {X 0,Y 594.433,Z 621.539,A -85,B 0,C 180,E1 -1003.394,E2 -1003.394} C_VEL
LIN {X 0,Y 594.524,Z 599.712,A -85,B 0,C 180,E1 -1006.304,E2 -1006.304} C_VEL
LIN {X 0,Y 594.625,Z 579.051,A -85,B 0,C 180,E1 -1009.098,E2 -1009.098} C_VEL
LIN {X 0,Y 594.769,Z 559.01,A -85,B 0,C 180,E1 -1011.851,E2 -1011.851} C_VEL
LIN {X 0,Y 594.866,Z 539.851,A -85,B 0,C 180,E1 -1014.534,E2 -1014.534} C_VEL
LIN {X 0,Y 594.868,Z 528.748,A -85,B 0,C 180,E1 -1016.117,E2 -1016.117} C_VEL
LIN {X 0,Y 594.398,Z 526.445,A -85,B 0,C 180,E1 -1016.484,E2 -1016.484} C_VEL
LIN {X 0,Y 594.382,Z 526.448,A -85,B 0,C 180,E1 -1018.997,E2 -1018.997} C_VEL
LIN {X 0,Y 594.392,Z 526.443,A -85,B 0,C 180,E1 -1021.644,E2 -1021.644} C_VEL
LIN {X 0,Y 594.396,Z 526.44,A -85,B 0,C 180,E1 -1024.578,E2 -1024.578} C_VEL
LIN {X 0,Y 594.385,Z 526.447,A -85,B 0,C 180,E1 -1027.085,E2 -1027.085} C_VEL
LIN {X 0,Y 594.373,Z 526.444,A -85,B 0,C 180,E1 -1029.774,E2 -1029.774} C_VEL
LIN {X 0,Y 594.365,Z 526.442,A -85,B 0,C 180,E1 -1032.374,E2 -1032.374} C_VEL
LIN {X 0,Y 594.357,Z 526.45,A -85,B 0,C 180,E1 -1035.19,E2 -1035.19} C_VEL
LIN {X 0,Y 594.383,Z 526.446,A -85,B 0,C 180,E1 -1037.626,E2 -1037.626} C_VEL
LIN {X 0,Y 594.389,Z 526.439,A -85,B 0,C 180,E1 -1040.32,E2 -1040.32} C_VEL
LIN {X 0,Y 594.383,Z 526.443,A -85,B 0,C 180,E1 -1042.913,E2 -1042.913} C_VEL
LIN {X 0,Y 594.392,Z 526.443,A -85,B 0,C 180,E1 -1045.002,E2 -1045.002} C_VEL
LIN {X 0,Y 594.739,Z 529.7,A -85,B 0,C 180,E1 -1045.057,E2 -1045.057} C_VEL
LIN {X 0,Y 594.639,Z 610.417,A -85,B 0,C 180,E1 -1046.054,E2 -1046.054} C_VEL
LIN {X 0,Y 594.595,Z 624.007,A -85,B 0,C 180,E1 -1046.367,E2 -1046.367} C_VEL
LIN {X 0,Y 594.568,Z 636.731,A -85,B 0,C 180,E1 -1046.809,E2 -1046.809} C_VEL
LIN {X 0,Y 594.488,Z 648.404,A -85,B 0,C 180,E1 -1047.359,E2 -1047.359} C_VEL
LIN {X 0,Y 594.437,Z 659.101,A -85,B 0,C 180,E1 -1047.996,E2 -1047.996} C_VEL
LIN {X 0,Y 594.406,Z 669.296,A -85,B 0,C 180,E1 -1048.751,E2 -1048.751} C_VEL
LIN {X 0,Y 594.353,Z 679.395,A -85,B 0,C 180,E1 -1049.675,E2 -1049.675} C_VEL
LIN {X 0,Y 594.313,Z 687.639,A -85,B 0,C 180,E1 -1050.61,E2 -1050.61} C_VEL
LIN {X 0,Y 594.286,Z 694.702,A -85,B 0,C 180,E1 -1051.59,E2 -1051.59} C_VEL
LIN {X 0,Y 594.261,Z 700.229,A -85,B 0,C 180,E1 -1052.533,E2 -1052.533} C_VEL
LIN {X 0,Y 594.287,Z 705.512,A -85,B 0,C 180,E1 -1053.675,E2 -1053.675} C_VEL
LIN {X 0,Y 594.237,Z 709.399,A -85,B 0,C 180,E1 -1054.8,E2 -1054.8} C_VEL
LIN {X 0,Y 594.231,Z 711.374,A -85,B 0,C 180,E1 -1055.597,E2 -1055.597} C_VEL
LIN {X 0,Y 594.223,Z 712.654,A -85,B 0,C 180,E1 -1056.289,E2 -1056.289} C_VEL
LIN {X 0,Y 594.249,Z 713.731,A -85,B 0,C 180,E1 -1057.288,E2 -1057.288} C_VEL
LIN {X 0,Y 594.222,Z 713.894,A -85,B 0,C 180,E1 -1058.491,E2 -1058.491} C_VEL
LIN {X 0,Y 594.25,Z 713.391,A -85,B 0,C 180,E1 -1059.219,E2 -1059.219} C_VEL
LIN {X 0,Y 594.218,Z 712.428,A -85,B 0,C 180,E1 -1059.941,E2 -1059.941} C_VEL
LIN {X 0,Y 594.24,Z 709.903,A -85,B 0,C 180,E1 -1061.107,E2 -1061.107} C_VEL
LIN {X 0,Y 594.253,Z 706.765,A -85,B 0,C 180,E1 -1062.092,E2 -1062.092} C_VEL
LIN {X 0,Y 594.268,Z 701.487,A -85,B 0,C 180,E1 -1063.317,E2 -1063.317} C_VEL
LIN {X 0,Y 594.282,Z 695.394,A -85,B 0,C 180,E1 -1064.393,E2 -1064.393} C_VEL
LIN {X 0,Y 594.34,Z 687.904,A -85,B 0,C 180,E1 -1065.447,E2 -1065.447} C_VEL
LIN {X 0,Y 594.375,Z 678.619,A -85,B 0,C 180,E1 -1066.495,E2 -1066.495} C_VEL
LIN {X 0,Y 594.411,Z 668.974,A -85,B 0,C 180,E1 -1067.365,E2 -1067.365} C_VEL
LIN {X 0,Y 594.455,Z 658.301,A -85,B 0,C 180,E1 -1068.146,E2 -1068.146} C_VEL
LIN {X 0,Y 594.517,Z 647.084,A -85,B 0,C 180,E1 -1068.802,E2 -1068.802} C_VEL
LIN {X 0,Y 594.573,Z 634.813,A -85,B 0,C 180,E1 -1069.357,E2 -1069.357} C_VEL
LIN {X 0,Y 594.617,Z 621.682,A -85,B 0,C 180,E1 -1069.788,E2 -1069.788} C_VEL
LIN {X 0,Y 594.655,Z 609.783,A -85,B 0,C 180,E1 -1070.047,E2 -1070.047} C_VEL
LIN {X 0,Y 594.591,Z 527.455,A -85,B 0,C 180,E1 -1071.063,E2 -1071.063} C_VEL
LIN {X 0,Y 594.395,Z 526.443,A -85,B 0,C 180,E1 -1071.115,E2 -1071.115} C_VEL
LIN {X 0,Y 594.38,Z 526.441,A -85,B 0,C 180,E1 -1073.891,E2 -1073.891} C_VEL
LIN {X 0,Y 594.384,Z 526.45,A -85,B 0,C 180,E1 -1076.611,E2 -1076.611} C_VEL
LIN {X 0,Y 594.419,Z 526.437,A -85,B 0,C 180,E1 -1079.323,E2 -1079.323} C_VEL
LIN {X 0,Y 594.387,Z 526.441,A -85,B 0,C 180,E1 -1082.033,E2 -1082.033} C_VEL
LIN {X 0,Y 594.399,Z 526.448,A -85,B 0,C 180,E1 -1084.748,E2 -1084.748} C_VEL
LIN {X 0,Y 594.393,Z 526.439,A -85,B 0,C 180,E1 -1087.473,E2 -1087.473} C_VEL
LIN {X 0,Y 594.391,Z 526.441,A -85,B 0,C 180,E1 -1090.216,E2 -1090.216} C_VEL
LIN {X 0,Y 594.363,Z 526.449,A -85,B 0,C 180,E1 -1092.983,E2 -1092.983} C_VEL
LIN {X 0,Y 594.362,Z 526.442,A -85,B 0,C 180,E1 -1095.781,E2 -1095.781} C_VEL
LIN {X 0,Y 594.381,Z 526.448,A -85,B 0,C 180,E1 -1098.618,E2 -1098.618} C_VEL
LIN {X 0,Y 594.36,Z 526.443,A -85,B 0,C 180,E1 -1101.504,E2 -1101.504} C_VEL
LIN {X 0,Y 594.379,Z 526.445,A -85,B 0,C 180,E1 -1104.447,E2 -1104.447} C_VEL
LIN {X 0,Y 594.382,Z 526.449,A -85,B 0,C 180,E1 -1106.7,E2 -1106.7} C_VEL
LIN {X 0,Y 594.378,Z 526.448,A -85,B 0,C 180,E1 -1108.999,E2 -1108.999} C_VEL
LIN {X 0,Y 594.385,Z 526.44,A -85,B 0,C 180,E1 -1111.646,E2 -1111.646} C_VEL
LIN {X 0,Y 594.395,Z 526.445,A -85,B 0,C 180,E1 -1114.579,E2 -1114.579} C_VEL
LIN {X 0,Y 594.383,Z 526.446,A -85,B 0,C 180,E1 -1117.087,E2 -1117.087} C_VEL
LIN {X 0,Y 594.374,Z 526.441,A -85,B 0,C 180,E1 -1119.776,E2 -1119.776} C_VEL
LIN {X 0,Y 594.384,Z 526.443,A -85,B 0,C 180,E1 -1122.374,E2 -1122.374} C_VEL
LIN {X 0,Y 594.357,Z 526.448,A -85,B 0,C 180,E1 -1125.192,E2 -1125.192} C_VEL
LIN {X 0,Y 594.365,Z 526.443,A -85,B 0,C 180,E1 -1127.626,E2 -1127.626} C_VEL
LIN {X 0,Y 594.391,Z 526.441,A -85,B 0,C 180,E1 -1130.322,E2 -1130.322} C_VEL
LIN {X 0,Y 594.385,Z 526.45,A -85,B 0,C 180,E1 -1132.915,E2 -1132.915} C_VEL
LIN {X 0,Y 594.383,Z 526.44,A -85,B 0,C 180,E1 -1135.862,E2 -1135.862} C_VEL
LIN {X 0,Y 594.389,Z 526.446,A -85,B 0,C 180,E1 -1138.652,E2 -1138.652} C_VEL
LIN {X 0,Y 594.383,Z 526.45,A -85,B 0,C 180,E1 -1141.043,E2 -1141.043} C_VEL
LIN {X 0,Y 594.389,Z 526.476,A -85,B 0,C 180,E1 -1143.381,E2 -1143.381} C_VEL
LIN {X 0,Y 595.214,Z 531.359,A -85,B 0,C 180,E1 -1143.968,E2 -1143.968} C_VEL
LIN {X 0,Y 595.016,Z 556.035,A -85,B 0,C 180,E1 -1146.692,E2 -1146.692} C_VEL
LIN {X 0,Y 594.856,Z 581.25,A -85,B 0,C 180,E1 -1149.423,E2 -1149.423} C_VEL
LIN {X 0,Y 594.703,Z 608.145,A -85,B 0,C 180,E1 -1152.285,E2 -1152.285} C_VEL
LIN {X 0,Y 594.557,Z 635.041,A -85,B 0,C 180,E1 -1155.103,E2 -1155.103} C_VEL
LIN {X 0,Y 594.523,Z 649.75,A -85,B 0,C 180,E1 -1156.63,E2 -1156.63} C_VEL
LIN {X 0,Y 594.761,Z 655.785,A -85,B 0,C 180,E1 -1156.722,E2 -1156.722} C_VEL
LIN {X 0,Y 594.678,Z 759.987,A -85,B 0,C 180,E1 -1158,E2 -1158} C_VEL
LIN {X 0,Y 594.641,Z 773.242,A -85,B 0,C 180,E1 -1158.302,E2 -1158.302} C_VEL
LIN {X 0,Y 594.58,Z 785.59,A -85,B 0,C 180,E1 -1158.719,E2 -1158.719} C_VEL
LIN {X 0,Y 594.538,Z 797.647,A -85,B 0,C 180,E1 -1159.271,E2 -1159.271} C_VEL
LIN {X 0,Y 594.472,Z 809.21,A -85,B 0,C 180,E1 -1159.958,E2 -1159.958} C_VEL
LIN {X 0,Y 594.413,Z 819.604,A -85,B 0,C 180,E1 -1160.73,E2 -1160.73} C_VEL
LIN {X 0,Y 594.383,Z 828.119,A -85,B 0,C 180,E1 -1161.501,E2 -1161.501} C_VEL
LIN {X 0,Y 594.347,Z 835.966,A -85,B 0,C 180,E1 -1162.356,E2 -1162.356} C_VEL
LIN {X 0,Y 594.282,Z 843.816,A -85,B 0,C 180,E1 -1163.409,E2 -1163.409} C_VEL
LIN {X 0,Y 594.289,Z 850.684,A -85,B 0,C 180,E1 -1164.572,E2 -1164.572} C_VEL
LIN {X 0,Y 594.271,Z 855.374,A -85,B 0,C 180,E1 -1165.592,E2 -1165.592} C_VEL
LIN {X 0,Y 594.268,Z 858.959,A -85,B 0,C 180,E1 -1166.611,E2 -1166.611} C_VEL
LIN {X 0,Y 594.226,Z 860.811,A -85,B 0,C 180,E1 -1167.289,E2 -1167.289} C_VEL
LIN {X 0,Y 594.239,Z 862.203,A -85,B 0,C 180,E1 -1167.967,E2 -1167.967} C_VEL
LIN {X 0,Y 594.239,Z 863.784,A -85,B 0,C 180,E1 -1169.323,E2 -1169.323} C_VEL
LIN {X 0,Y 594.236,Z 864,A -85,B 0,C 180,E1 -1170.001,E2 -1170.001} C_VEL
LIN {X 0,Y 594.247,Z 863.184,A -85,B 0,C 180,E1 -1171.356,E2 -1171.356} C_VEL
LIN {X 0,Y 594.239,Z 862.201,A -85,B 0,C 180,E1 -1172.034,E2 -1172.034} C_VEL
LIN {X 0,Y 594.226,Z 860.808,A -85,B 0,C 180,E1 -1172.712,E2 -1172.712} C_VEL
LIN {X 0,Y 594.289,Z 857.894,A -85,B 0,C 180,E1 -1173.73,E2 -1173.73} C_VEL
LIN {X 0,Y 594.241,Z 853.948,A -85,B 0,C 180,E1 -1174.749,E2 -1174.749} C_VEL
LIN {X 0,Y 594.304,Z 847.874,A -85,B 0,C 180,E1 -1175.94,E2 -1175.94} C_VEL
LIN {X 0,Y 594.308,Z 841.233,A -85,B 0,C 180,E1 -1176.962,E2 -1176.962} C_VEL
LIN {X 0,Y 594.359,Z 832.986,A -85,B 0,C 180,E1 -1177.987,E2 -1177.987} C_VEL
LIN {X 0,Y 594.382,Z 824.532,A -85,B 0,C 180,E1 -1178.843,E2 -1178.843} C_VEL
LIN {X 0,Y 594.423,Z 814.088,A -85,B 0,C 180,E1 -1179.7,E2 -1179.7} C_VEL
LIN {X 0,Y 594.489,Z 803.751,A -85,B 0,C 180,E1 -1180.387,E2 -1180.387} C_VEL
LIN {X 0,Y 594.56,Z 792.698,A -85,B 0,C 180,E1 -1180.974,E2 -1180.974} C_VEL
LIN {X 0,Y 594.602,Z 780.696,A -85,B 0,C 180,E1 -1181.464,E2 -1181.464} C_VEL
LIN {X 0,Y 594.639,Z 767.337,A -85,B 0,C 180,E1 -1181.851,E2 -1181.851} C_VEL
LIN {X 0,Y 594.681,Z 754.055,A -85,B 0,C 180,E1 -1182.088,E2 -1182.088} C_VEL
LIN {X 0,Y 594.686,Z 652.112,A -85,B 0,C 180,E1 -1183.324,E2 -1183.324} C_VEL
LIN {X 0,Y 594.487,Z 650.468,A -85,B 0,C 180,E1 -1183.372,E2 -1183.372} C_VEL
LIN {X 0,Y 594.566,Z 626.829,A -85,B 0,C 180,E1 -1186.128,E2 -1186.128} C_VEL
LIN {X 0,Y 594.698,Z 603.418,A -85,B 0,C 180,E1 -1188.893,E2 -1188.893} C_VEL
LIN {X 0,Y 594.87,Z 580.302,A -85,B 0,C 180,E1 -1191.666,E2 -1191.666} C_VEL
LIN {X 0,Y 595.028,Z 556.577,A -85,B 0,C 180,E1 -1194.568,E2 -1194.568} C_VEL
LIN {X 0,Y 595.204,Z 532.753,A -85,B 0,C 180,E1 -1197.549,E2 -1197.549} C_VEL
LIN {X 0,Y 594.963,Z 529.018,A -85,B 0,C 180,E1 -1198.037,E2 -1198.037} C_VEL
LIN {X 0,Y 594.379,Z 526.448,A -85,B 0,C 180,E1 -1198.419,E2 -1198.419} C_VEL
LIN {X 0,Y 594.394,Z 526.443,A -85,B 0,C 180,E1 -1201.349,E2 -1201.349} C_VEL
LIN {X 0,Y 594.386,Z 526.44,A -85,B 0,C 180,E1 -1204.139,E2 -1204.139} C_VEL
LIN {X 0,Y 594.387,Z 526.449,A -85,B 0,C 180,E1 -1207.087,E2 -1207.087} C_VEL
LIN {X 0,Y 594.379,Z 526.441,A -85,B 0,C 180,E1 -1209.774,E2 -1209.774} C_VEL
LIN {X 0,Y 594.368,Z 526.442,A -85,B 0,C 180,E1 -1212.375,E2 -1212.375} C_VEL
LIN {X 0,Y 594.366,Z 526.452,A -85,B 0,C 180,E1 -1215.191,E2 -1215.191} C_VEL
LIN {X 0,Y 594.373,Z 526.443,A -85,B 0,C 180,E1 -1217.625,E2 -1217.625} C_VEL
LIN {X 0,Y 594.392,Z 526.439,A -85,B 0,C 180,E1 -1220.321,E2 -1220.321} C_VEL
LIN {X 0,Y 594.389,Z 526.444,A -85,B 0,C 180,E1 -1222.913,E2 -1222.913} C_VEL
LIN {X 0,Y 594.386,Z 526.441,A -85,B 0,C 180,E1 -1225.861,E2 -1225.861} C_VEL
LIN {X 0,Y 594.379,Z 526.441,A -85,B 0,C 180,E1 -1228.65,E2 -1228.65} C_VEL
LIN {X 0,Y 594.384,Z 526.445,A -85,B 0,C 180,E1 -1231.042,E2 -1231.042} C_VEL
LIN {X 0,Y 594.385,Z 526.44,A -85,B 0,C 180,E1 -1233.977,E2 -1233.977} C_VEL
LIN {X 0,Y 594.39,Z 526.438,A -85,B 0,C 180,E1 -1236.296,E2 -1236.296} C_VEL
LIN {X 0,Y 594.409,Z 526.444,A -85,B 0,C 180,E1 -1239.225,E2 -1239.225} C_VEL
LIN {X 0,Y 594.356,Z 526.443,A -85,B 0,C 180,E1 -1242.095,E2 -1242.095} C_VEL
LIN {X 0,Y 594.366,Z 526.442,A -85,B 0,C 180,E1 -1244.219,E2 -1244.219} C_VEL
LIN {X 0,Y 594.367,Z 526.444,A -85,B 0,C 180,E1 -1247.017,E2 -1247.017} C_VEL
LIN {X 0,Y 594.397,Z 526.444,A -85,B 0,C 180,E1 -1249.784,E2 -1249.784} C_VEL
LIN {X 0,Y 594.392,Z 526.438,A -85,B 0,C 180,E1 -1252.527,E2 -1252.527} C_VEL
LIN {X 0,Y 594.399,Z 526.442,A -85,B 0,C 180,E1 -1255.252,E2 -1255.252} C_VEL
LIN {X 0,Y 594.396,Z 526.443,A -85,B 0,C 180,E1 -1257.967,E2 -1257.967} C_VEL
LIN {X 0,Y 594.421,Z 526.435,A -85,B 0,C 180,E1 -1260.677,E2 -1260.677} C_VEL
LIN {X 0,Y 594.378,Z 526.445,A -85,B 0,C 180,E1 -1263.389,E2 -1263.389} C_VEL
LIN {X 0,Y 594.373,Z 526.445,A -85,B 0,C 180,E1 -1266.109,E2 -1266.109} C_VEL
LIN {X 0,Y 594.398,Z 526.438,A -85,B 0,C 180,E1 -1268.842,E2 -1268.842} C_VEL
LIN {X 0,Y 594.393,Z 526.445,A -85,B 0,C 180,E1 -1271.596,E2 -1271.596} C_VEL
LIN {X 0,Y 594.388,Z 526.442,A -85,B 0,C 180,E1 -1274.377,E2 -1274.377} C_VEL
LIN {X 0,Y 594.358,Z 526.445,A -85,B 0,C 180,E1 -1275.33,E2 -1275.33} C_VEL
LIN {X 0,Y 593.69,Z 526.537,A -85,B 0,C 180,E1 -1275.896,E2 -1275.896} C_VEL
LIN {X 0,Y 590.837,Z 526.893,A -85,B 0,C 180,E1 -1276.814,E2 -1276.814} C_VEL
LIN {X 0,Y 588.432,Z 527.191,A -85,B 0,C 180,E1 -1277.553,E2 -1277.553} C_VEL
LIN {X 0,Y 587.405,Z 527.315,A -85,B 0,C 180,E1 -1278.123,E2 -1278.123} C_VEL
LIN {X 0,Y 587.324,Z 527.322,A -85,B 0,C 180,E1 -1278.316,E2 -1278.316} C_VEL
LIN {X 0,Y 587.33,Z 527.318,A -85,B 0,C 180,E1 -1281.038,E2 -1281.038} C_VEL
LIN {X 0,Y 587.323,Z 527.32,A -85,B 0,C 180,E1 -1283.259,E2 -1283.259} C_VEL
LIN {X 0,Y 587.333,Z 527.32,A -85,B 0,C 180,E1 -1285.517,E2 -1285.517} C_VEL
LIN {X 0,Y 587.348,Z 527.323,A -85,B 0,C 180,E1 -1287.818,E2 -1287.818} C_VEL
LIN {X 0,Y 587.337,Z 527.32,A -85,B 0,C 180,E1 -1290.51,E2 -1290.51} C_VEL
LIN {X 0,Y 587.333,Z 527.319,A -85,B 0,C 180,E1 -1293.397,E2 -1293.397} C_VEL
LIN {X 0,Y 587.291,Z 527.329,A -85,B 0,C 180,E1 -1295.9,E2 -1295.9} C_VEL
LIN {X 0,Y 587.335,Z 527.323,A -85,B 0,C 180,E1 -1298.479,E2 -1298.479} C_VEL
LIN {X 0,Y 587.337,Z 527.318,A -85,B 0,C 180,E1 -1301.157,E2 -1301.157} C_VEL
LIN {X 0,Y 587.337,Z 527.326,A -85,B 0,C 180,E1 -1304.114,E2 -1304.114} C_VEL
LIN {X 0,Y 587.314,Z 527.319,A -85,B 0,C 180,E1 -1306.994,E2 -1306.994} C_VEL
LIN {X 0,Y 587.313,Z 527.323,A -85,B 0,C 180,E1 -1309.746,E2 -1309.746} C_VEL
LIN {X 0,Y 587.344,Z 527.326,A -85,B 0,C 180,E1 -1312.392,E2 -1312.392} C_VEL
LIN {X 0,Y 587.355,Z 527.316,A -85,B 0,C 180,E1 -1315.652,E2 -1315.652} C_VEL
LIN {X 0,Y 587.344,Z 527.325,A -85,B 0,C 180,E1 -1318.231,E2 -1318.231} C_VEL
LIN {X 0,Y 587.353,Z 527.32,A -85,B 0,C 180,E1 -1320.867,E2 -1320.867} C_VEL
LIN {X 0,Y 587.363,Z 527.317,A -85,B 0,C 180,E1 -1323.819,E2 -1323.819} C_VEL
LIN {X 0,Y 587.36,Z 527.451,A -85,B 0,C 180,E1 -1324.982,E2 -1324.982} C_VEL
LIN {X 0,Y 588.091,Z 530.888,A -85,B 0,C 180,E1 -1325.456,E2 -1325.456} C_VEL
LIN {X 0,Y 587.978,Z 548.577,A -85,B 0,C 180,E1 -1327.697,E2 -1327.697} C_VEL
LIN {X 0,Y 587.76,Z 571.694,A -85,B 0,C 180,E1 -1330.572,E2 -1330.572} C_VEL
LIN {X 0,Y 587.61,Z 594.139,A -85,B 0,C 180,E1 -1333.318,E2 -1333.318} C_VEL
LIN {X 0,Y 587.467,Z 619.126,A -85,B 0,C 180,E1 -1336.333,E2 -1336.333} C_VEL
LIN {X 0,Y 587.509,Z 621.14,A -85,B 0,C 180,E1 -1336.543,E2 -1336.543} C_VEL
LIN {X 0,Y 587.825,Z 627.397,A -85,B 0,C 180,E1 -1336.628,E2 -1336.628} C_VEL
LIN {X 0,Y 587.721,Z 729.832,A -85,B 0,C 180,E1 -1337.898,E2 -1337.898} C_VEL
LIN {X 0,Y 587.695,Z 743.185,A -85,B 0,C 180,E1 -1338.204,E2 -1338.204} C_VEL
LIN {X 0,Y 587.611,Z 755.792,A -85,B 0,C 180,E1 -1338.636,E2 -1338.636} C_VEL
LIN {X 0,Y 587.542,Z 768.405,A -85,B 0,C 180,E1 -1339.228,E2 -1339.228} C_VEL
LIN {X 0,Y 587.461,Z 779.818,A -85,B 0,C 180,E1 -1339.923,E2 -1339.923} C_VEL
LIN {X 0,Y 587.383,Z 790.098,A -85,B 0,C 180,E1 -1340.704,E2 -1340.704} C_VEL
LIN {X 0,Y 587.341,Z 799.369,A -85,B 0,C 180,E1 -1341.571,E2 -1341.571} C_VEL
LIN {X 0,Y 587.26,Z 808.339,A -85,B 0,C 180,E1 -1342.608,E2 -1342.608} C_VEL
LIN {X 0,Y 587.199,Z 815.435,A -85,B 0,C 180,E1 -1343.624,E2 -1343.624} C_VEL
LIN {X 0,Y 587.211,Z 820.445,A -85,B 0,C 180,E1 -1344.505,E2 -1344.505} C_VEL
LIN {X 0,Y 587.188,Z 825.187,A -85,B 0,C 180,E1 -1345.538,E2 -1345.538} C_VEL
LIN {X 0,Y 587.193,Z 828.818,A -85,B 0,C 180,E1 -1346.569,E2 -1346.569} C_VEL
LIN {X 0,Y 587.131,Z 830.692,A -85,B 0,C 180,E1 -1347.255,E2 -1347.255} C_VEL
LIN {X 0,Y 587.139,Z 832.127,A -85,B 0,C 180,E1 -1347.942,E2 -1347.942} C_VEL
LIN {X 0,Y 587.14,Z 833.753,A -85,B 0,C 180,E1 -1349.314,E2 -1349.314} C_VEL
LIN {X 0,Y 587.137,Z 833.996,A -85,B 0,C 180,E1 -1349.999,E2 -1349.999} C_VEL
LIN {X 0,Y 587.14,Z 833.815,A -85,B 0,C 180,E1 -1350.685,E2 -1350.685} C_VEL
LIN {X 0,Y 587.14,Z 832.274,A -85,B 0,C 180,E1 -1352.057,E2 -1352.057} C_VEL
LIN {X 0,Y 587.132,Z 830.916,A -85,B 0,C 180,E1 -1352.744,E2 -1352.744} C_VEL
LIN {X 0,Y 587.213,Z 828.041,A -85,B 0,C 180,E1 -1353.774,E2 -1353.774} C_VEL
LIN {X 0,Y 587.147,Z 824.143,A -85,B 0,C 180,E1 -1354.806,E2 -1354.806} C_VEL
LIN {X 0,Y 587.229,Z 819.112,A -85,B 0,C 180,E1 -1355.838,E2 -1355.838} C_VEL
LIN {X 0,Y 587.229,Z 812.784,A -85,B 0,C 180,E1 -1356.873,E2 -1356.873} C_VEL
LIN {X 0,Y 587.287,Z 804.878,A -85,B 0,C 180,E1 -1357.909,E2 -1357.909} C_VEL
LIN {X 0,Y 587.343,Z 795.023,A -85,B 0,C 180,E1 -1358.948,E2 -1358.948} C_VEL
LIN {X 0,Y 587.415,Z 784.71,A -85,B 0,C 180,E1 -1359.816,E2 -1359.816} C_VEL
LIN {X 0,Y 587.526,Z 773.096,A -85,B 0,C 180,E1 -1360.597,E2 -1360.597} C_VEL
LIN {X 0,Y 587.599,Z 762.008,A -85,B 0,C 180,E1 -1361.183,E2 -1361.183} C_VEL
LIN {X 0,Y 587.627,Z 749.596,A -85,B 0,C 180,E1 -1361.685,E2 -1361.685} C_VEL
LIN {X 0,Y 587.727,Z 736.554,A -85,B 0,C 180,E1 -1362.057,E2 -1362.057} C_VEL
LIN {X 0,Y 587.742,Z 724.228,A -85,B 0,C 180,E1 -1362.275,E2 -1362.275} C_VEL
LIN {X 0,Y 587.742,Z 623.85,A -85,B 0,C 180,E1 -1363.508,E2 -1363.508} C_VEL
LIN {X 0,Y 587.419,Z 621.535,A -85,B 0,C 180,E1 -1363.557,E2 -1363.557} C_VEL
LIN {X 0,Y 587.547,Z 599.708,A -85,B 0,C 180,E1 -1366.503,E2 -1366.503} C_VEL
LIN {X 0,Y 587.685,Z 578.395,A -85,B 0,C 180,E1 -1369.423,E2 -1369.423} C_VEL
LIN {X 0,Y 587.904,Z 557.692,A -85,B 0,C 180,E1 -1372.305,E2 -1372.305} C_VEL
LIN {X 0,Y 588.074,Z 536.683,A -85,B 0,C 180,E1 -1375.292,E2 -1375.292} C_VEL
LIN {X 0,Y 587.885,Z 529.889,A -85,B 0,C 180,E1 -1376.284,E2 -1376.284} C_VEL
LIN {X 0,Y 587.373,Z 527.322,A -85,B 0,C 180,E1 -1376.706,E2 -1376.706} C_VEL
LIN {X 0,Y 587.346,Z 527.325,A -85,B 0,C 180,E1 -1379.378,E2 -1379.378} C_VEL
LIN {X 0,Y 587.355,Z 527.318,A -85,B 0,C 180,E1 -1381.837,E2 -1381.837} C_VEL
LIN {X 0,Y 587.355,Z 527.316,A -85,B 0,C 180,E1 -1384.348,E2 -1384.348} C_VEL
LIN {X 0,Y 587.351,Z 527.318,A -85,B 0,C 180,E1 -1386.745,E2 -1386.745} C_VEL
LIN {X 0,Y 587.343,Z 527.326,A -85,B 0,C 180,E1 -1389.358,E2 -1389.358} C_VEL
LIN {X 0,Y 587.329,Z 527.319,A -85,B 0,C 180,E1 -1392.107,E2 -1392.107} C_VEL
LIN {X 0,Y 587.31,Z 527.326,A -85,B 0,C 180,E1 -1395.088,E2 -1395.088} C_VEL
LIN {X 0,Y 587.346,Z 527.319,A -85,B 0,C 180,E1 -1397.927,E2 -1397.927} C_VEL
LIN {X 0,Y 587.343,Z 527.318,A -85,B 0,C 180,E1 -1400.64,E2 -1400.64} C_VEL
LIN {X 0,Y 587.348,Z 527.326,A -85,B 0,C 180,E1 -1403.29,E2 -1403.29} C_VEL
LIN {X 0,Y 587.348,Z 527.454,A -85,B 0,C 180,E1 -1404.863,E2 -1404.863} C_VEL
LIN {X 0,Y 587.803,Z 529.138,A -85,B 0,C 180,E1 -1404.894,E2 -1404.894} C_VEL
LIN {X 0,Y 587.701,Z 610.101,A -85,B 0,C 180,E1 -1405.906,E2 -1405.906} C_VEL
LIN {X 0,Y 587.654,Z 623.061,A -85,B 0,C 180,E1 -1406.2,E2 -1406.2} C_VEL
LIN {X 0,Y 587.613,Z 635.427,A -85,B 0,C 180,E1 -1406.621,E2 -1406.621} C_VEL
LIN {X 0,Y 587.513,Z 646.986,A -85,B 0,C 180,E1 -1407.153,E2 -1407.153} C_VEL
LIN {X 0,Y 587.458,Z 658.308,A -85,B 0,C 180,E1 -1407.824,E2 -1407.824} C_VEL
LIN {X 0,Y 587.385,Z 668.025,A -85,B 0,C 180,E1 -1408.535,E2 -1408.535} C_VEL
LIN {X 0,Y 587.339,Z 678.561,A -85,B 0,C 180,E1 -1409.487,E2 -1409.487} C_VEL
LIN {X 0,Y 587.272,Z 686.848,A -85,B 0,C 180,E1 -1410.419,E2 -1410.419} C_VEL
LIN {X 0,Y 587.205,Z 693.954,A -85,B 0,C 180,E1 -1411.397,E2 -1411.397} C_VEL
LIN {X 0,Y 587.196,Z 699.522,A -85,B 0,C 180,E1 -1412.333,E2 -1412.333} C_VEL
LIN {X 0,Y 587.196,Z 704.307,A -85,B 0,C 180,E1 -1413.331,E2 -1413.331} C_VEL
LIN {X 0,Y 587.143,Z 708.51,A -85,B 0,C 180,E1 -1414.474,E2 -1414.474} C_VEL
LIN {X 0,Y 587.13,Z 711.147,A -85,B 0,C 180,E1 -1415.464,E2 -1415.464} C_VEL
LIN {X 0,Y 587.116,Z 713.249,A -85,B 0,C 180,E1 -1416.732,E2 -1416.732} C_VEL
LIN {X 0,Y 587.147,Z 713.834,A -85,B 0,C 180,E1 -1417.478,E2 -1417.478} C_VEL
LIN {X 0,Y 587.138,Z 713.967,A -85,B 0,C 180,E1 -1418.218,E2 -1418.218} C_VEL
LIN {X 0,Y 587.162,Z 713.602,A -85,B 0,C 180,E1 -1419.002,E2 -1419.002} C_VEL
LIN {X 0,Y 587.147,Z 712.834,A -85,B 0,C 180,E1 -1419.688,E2 -1419.688} C_VEL
LIN {X 0,Y 587.148,Z 710.247,A -85,B 0,C 180,E1 -1421.011,E2 -1421.011} C_VEL
LIN {X 0,Y 587.172,Z 706.451,A -85,B 0,C 180,E1 -1422.229,E2 -1422.229} C_VEL
LIN {X 0,Y 587.175,Z 701.855,A -85,B 0,C 180,E1 -1423.306,E2 -1423.306} C_VEL
LIN {X 0,Y 587.198,Z 695.962,A -85,B 0,C 180,E1 -1424.378,E2 -1424.378} C_VEL
LIN {X 0,Y 587.262,Z 689.947,A -85,B 0,C 180,E1 -1425.267,E2 -1425.267} C_VEL
LIN {X 0,Y 587.279,Z 682.741,A -85,B 0,C 180,E1 -1426.152,E2 -1426.152} C_VEL
LIN {X 0,Y 587.348,Z 674.051,A -85,B 0,C 180,E1 -1427.035,E2 -1427.035} C_VEL
LIN {X 0,Y 587.408,Z 663.4,A -85,B 0,C 180,E1 -1427.914,E2 -1427.914} C_VEL
LIN {X 0,Y 587.511,Z 652.538,A -85,B 0,C 180,E1 -1428.63,E2 -1428.63} C_VEL
LIN {X 0,Y 587.589,Z 640.938,A -85,B 0,C 180,E1 -1429.229,E2 -1429.229} C_VEL
LIN {X 0,Y 587.636,Z 630.067,A -85,B 0,C 180,E1 -1429.665,E2 -1429.665} C_VEL
LIN {X 0,Y 587.683,Z 618.273,A -85,B 0,C 180,E1 -1430.014,E2 -1430.014} C_VEL
LIN {X 0,Y 587.726,Z 605.715,A -85,B 0,C 180,E1 -1430.254,E2 -1430.254} C_VEL
LIN {X 0,Y 587.767,Z 528.979,A -85,B 0,C 180,E1 -1431.198,E2 -1431.198} C_VEL
LIN {X 0,Y 587.346,Z 527.32,A -85,B 0,C 180,E1 -1431.246,E2 -1431.246} C_VEL
LIN {X 0,Y 587.334,Z 527.319,A -85,B 0,C 180,E1 -1433.818,E2 -1433.818} C_VEL
LIN {X 0,Y 587.313,Z 527.322,A -85,B 0,C 180,E1 -1435.883,E2 -1435.883} C_VEL
LIN {X 0,Y 587.358,Z 527.316,A -85,B 0,C 180,E1 -1437.943,E2 -1437.943} C_VEL
LIN {X 0,Y 587.394,Z 527.322,A -85,B 0,C 180,E1 -1440.686,E2 -1440.686} C_VEL
LIN {X 0,Y 587.33,Z 527.319,A -85,B 0,C 180,E1 -1443.43,E2 -1443.43} C_VEL
LIN {X 0,Y 587.356,Z 527.316,A -85,B 0,C 180,E1 -1445.493,E2 -1445.493} C_VEL
LIN {X 0,Y 587.364,Z 527.317,A -85,B 0,C 180,E1 -1448.255,E2 -1448.255} C_VEL
LIN {X 0,Y 587.351,Z 527.32,A -85,B 0,C 180,E1 -1451.142,E2 -1451.142} C_VEL
LIN {X 0,Y 587.353,Z 527.319,A -85,B 0,C 180,E1 -1454.261,E2 -1454.261} C_VEL
LIN {X 0,Y 587.35,Z 527.317,A -85,B 0,C 180,E1 -1457.406,E2 -1457.406} C_VEL
LIN {X 0,Y 587.325,Z 527.322,A -85,B 0,C 180,E1 -1460.305,E2 -1460.305} C_VEL
LIN {X 0,Y 587.317,Z 527.323,A -85,B 0,C 180,E1 -1463.259,E2 -1463.259} C_VEL
LIN {X 0,Y 587.353,Z 527.317,A -85,B 0,C 180,E1 -1466.183,E2 -1466.183} C_VEL
LIN {X 0,Y 587.346,Z 527.321,A -85,B 0,C 180,E1 -1469.135,E2 -1469.135} C_VEL
LIN {X 0,Y 587.349,Z 527.316,A -85,B 0,C 180,E1 -1471.839,E2 -1471.839} C_VEL
LIN {X 0,Y 587.353,Z 527.319,A -85,B 0,C 180,E1 -1474.351,E2 -1474.351} C_VEL
LIN {X 0,Y 587.347,Z 527.326,A -85,B 0,C 180,E1 -1476.747,E2 -1476.747} C_VEL
LIN {X 0,Y 587.343,Z 527.319,A -85,B 0,C 180,E1 -1479.36,E2 -1479.36} C_VEL
LIN {X 0,Y 587.36,Z 527.316,A -85,B 0,C 180,E1 -1482.112,E2 -1482.112} C_VEL
LIN {X 0,Y 587.31,Z 527.328,A -85,B 0,C 180,E1 -1485.09,E2 -1485.09} C_VEL
LIN {X 0,Y 587.347,Z 527.317,A -85,B 0,C 180,E1 -1487.929,E2 -1487.929} C_VEL
LIN {X 0,Y 587.333,Z 527.326,A -85,B 0,C 180,E1 -1491.059,E2 -1491.059} C_VEL
LIN {X 0,Y 587.351,Z 527.32,A -85,B 0,C 180,E1 -1493.292,E2 -1493.292} C_VEL
LIN {X 0,Y 587.365,Z 527.315,A -85,B 0,C 180,E1 -1495.782,E2 -1495.782} C_VEL
LIN {X 0,Y 587.352,Z 527.318,A -85,B 0,C 180,E1 -1498.233,E2 -1498.233} C_VEL
LIN {X 0,Y 587.349,Z 527.327,A -85,B 0,C 180,E1 -1500.867,E2 -1500.867} C_VEL
LIN {X 0,Y 587.37,Z 527.46,A -85,B 0,C 180,E1 -1503.149,E2 -1503.149} C_VEL
LIN {X 0,Y 588.44,Z 532.501,A -85,B 0,C 180,E1 -1503.775,E2 -1503.775} C_VEL
LIN {X 0,Y 588.23,Z 556.035,A -85,B 0,C 180,E1 -1506.407,E2 -1506.407} C_VEL
LIN {X 0,Y 587.976,Z 581.25,A -85,B 0,C 180,E1 -1509.171,E2 -1509.171} C_VEL
LIN {X 0,Y 587.777,Z 608.145,A -85,B 0,C 180,E1 -1512.069,E2 -1512.069} C_VEL
LIN {X 0,Y 587.587,Z 633.36,A -85,B 0,C 180,E1 -1514.745,E2 -1514.745} C_VEL
LIN {X 0,Y 587.504,Z 649.75,A -85,B 0,C 180,E1 -1516.467,E2 -1516.467} C_VEL
LIN {X 0,Y 587.886,Z 653.996,A -85,B 0,C 180,E1 -1516.542,E2 -1516.542} C_VEL
LIN {X 0,Y 587.735,Z 759.986,A -85,B 0,C 180,E1 -1517.856,E2 -1517.856} C_VEL
LIN {X 0,Y 587.701,Z 772.482,A -85,B 0,C 180,E1 -1518.14,E2 -1518.14} C_VEL
LIN {X 0,Y 587.613,Z 785.769,A -85,B 0,C 180,E1 -1518.591,E2 -1518.591} C_VEL
LIN {X 0,Y 587.553,Z 797.646,A -85,B 0,C 180,E1 -1519.142,E2 -1519.142} C_VEL
LIN {X 0,Y 587.462,Z 809.211,A -85,B 0,C 180,E1 -1519.837,E2 -1519.837} C_VEL
LIN {X 0,Y 587.391,Z 819.605,A -85,B 0,C 180,E1 -1520.618,E2 -1520.618} C_VEL
LIN {X 0,Y 587.321,Z 828.12,A -85,B 0,C 180,E1 -1521.398,E2 -1521.398} C_VEL
LIN {X 0,Y 587.273,Z 835.966,A -85,B 0,C 180,E1 -1522.263,E2 -1522.263} C_VEL
LIN {X 0,Y 587.232,Z 842.475,A -85,B 0,C 180,E1 -1523.127,E2 -1523.127} C_VEL
LIN {X 0,Y 587.236,Z 848.87,A -85,B 0,C 180,E1 -1524.162,E2 -1524.162} C_VEL
LIN {X 0,Y 587.147,Z 853.952,A -85,B 0,C 180,E1 -1525.194,E2 -1525.194} C_VEL
LIN {X 0,Y 587.213,Z 857.898,A -85,B 0,C 180,E1 -1526.226,E2 -1526.226} C_VEL
LIN {X 0,Y 587.132,Z 860.811,A -85,B 0,C 180,E1 -1527.256,E2 -1527.256} C_VEL
LIN {X 0,Y 587.138,Z 862.202,A -85,B 0,C 180,E1 -1527.943,E2 -1527.943} C_VEL
LIN {X 0,Y 587.14,Z 863.785,A -85,B 0,C 180,E1 -1529.315,E2 -1529.315} C_VEL
LIN {X 0,Y 587.137,Z 864,A -85,B 0,C 180,E1 -1530.001,E2 -1530.001} C_VEL
LIN {X 0,Y 587.147,Z 863.184,A -85,B 0,C 180,E1 -1531.372,E2 -1531.372} C_VEL
LIN {X 0,Y 587.138,Z 862.2,A -85,B 0,C 180,E1 -1532.058,E2 -1532.058} C_VEL
LIN {X 0,Y 587.132,Z 860.807,A -85,B 0,C 180,E1 -1532.745,E2 -1532.745} C_VEL
LIN {X 0,Y 587.213,Z 857.894,A -85,B 0,C 180,E1 -1533.775,E2 -1533.775} C_VEL
LIN {X 0,Y 587.147,Z 853.948,A -85,B 0,C 180,E1 -1534.807,E2 -1534.807} C_VEL
LIN {X 0,Y 587.217,Z 847.875,A -85,B 0,C 180,E1 -1536.012,E2 -1536.012} C_VEL
LIN {X 0,Y 587.245,Z 841.233,A -85,B 0,C 180,E1 -1537.047,E2 -1537.047} C_VEL
LIN {X 0,Y 587.3,Z 832.986,A -85,B 0,C 180,E1 -1538.083,E2 -1538.083} C_VEL
LIN {X 0,Y 587.343,Z 824.532,A -85,B 0,C 180,E1 -1538.949,E2 -1538.949} C_VEL
LIN {X 0,Y 587.412,Z 814.089,A -85,B 0,C 180,E1 -1539.817,E2 -1539.817} C_VEL
LIN {X 0,Y 587.507,Z 803.751,A -85,B 0,C 180,E1 -1540.512,E2 -1540.512} C_VEL
LIN {X 0,Y 587.584,Z 791.797,A -85,B 0,C 180,E1 -1541.149,E2 -1541.149} C_VEL
LIN {X 0,Y 587.657,Z 779.585,A -85,B 0,C 180,E1 -1541.639,E2 -1541.639} C_VEL
LIN {X 0,Y 587.678,Z 766.422,A -85,B 0,C 180,E1 -1542.015,E2 -1542.015} C_VEL
LIN {X 0,Y 587.764,Z 754.055,A -85,B 0,C 180,E1 -1542.232,E2 -1542.232} C_VEL
LIN {X 0,Y 587.785,Z 652.894,A -85,B 0,C 180,E1 -1543.474,E2 -1543.474} C_VEL
LIN {X 0,Y 587.49,Z 650.468,A -85,B 0,C 180,E1 -1543.534,E2 -1543.534} C_VEL
LIN {X 0,Y 587.586,Z 626.83,A -85,B 0,C 180,E1 -1546.325,E2 -1546.325} C_VEL
LIN {X 0,Y 587.783,Z 604.123,A -85,B 0,C 180,E1 -1549.039,E2 -1549.039} C_VEL
LIN {X 0,Y 587.986,Z 580.302,A -85,B 0,C 180,E1 -1551.933,E2 -1551.933} C_VEL
LIN {X 0,Y 588.198,Z 557.486,A -85,B 0,C 180,E1 -1554.759,E2 -1554.759} C_VEL
LIN {X 0,Y 588.457,Z 533.775,A -85,B 0,C 180,E1 -1557.761,E2 -1557.761} C_VEL
LIN {X 0,Y 587.768,Z 529.274,A -85,B 0,C 180,E1 -1558.378,E2 -1558.378} C_VEL
LIN {X 0,Y 587.392,Z 527.32,A -85,B 0,C 180,E1 -1558.678,E2 -1558.678} C_VEL
LIN {X 0,Y 587.357,Z 527.316,A -85,B 0,C 180,E1 -1561.837,E2 -1561.837} C_VEL
LIN {X 0,Y 587.357,Z 527.317,A -85,B 0,C 180,E1 -1564.349,E2 -1564.349} C_VEL
LIN {X 0,Y 587.347,Z 527.318,A -85,B 0,C 180,E1 -1567.608,E2 -1567.608} C_VEL
LIN {X 0,Y 587.32,Z 527.32,A -85,B 0,C 180,E1 -1570.254,E2 -1570.254} C_VEL
LIN {X 0,Y 587.317,Z 527.33,A -85,B 0,C 180,E1 -1573.118,E2 -1573.118} C_VEL
LIN {X 0,Y 587.336,Z 527.318,A -85,B 0,C 180,E1 -1576.051,E2 -1576.051} C_VEL
LIN {X 0,Y 587.339,Z 527.323,A -85,B 0,C 180,E1 -1578.925,E2 -1578.925} C_VEL
LIN {X 0,Y 587.336,Z 527.322,A -85,B 0,C 180,E1 -1581.521,E2 -1581.521} C_VEL
LIN {X 0,Y 587.352,Z 527.315,A -85,B 0,C 180,E1 -1584.455,E2 -1584.455} C_VEL
LIN {X 0,Y 587.339,Z 527.321,A -85,B 0,C 180,E1 -1586.888,E2 -1586.888} C_VEL
LIN {X 0,Y 587.34,Z 527.324,A -85,B 0,C 180,E1 -1589.489,E2 -1589.489} C_VEL
LIN {X 0,Y 587.351,Z 527.316,A -85,B 0,C 180,E1 -1592.307,E2 -1592.307} C_VEL
LIN {X 0,Y 587.333,Z 527.317,A -85,B 0,C 180,E1 -1594.483,E2 -1594.483} C_VEL
LIN {X 0,Y 587.318,Z 527.325,A -85,B 0,C 180,E1 -1597.131,E2 -1597.131} C_VEL
LIN {X 0,Y 587.333,Z 527.323,A -85,B 0,C 180,E1 -1599.695,E2 -1599.695} C_VEL
LIN {X 0,Y 587.35,Z 527.314,A -85,B 0,C 180,E1 -1602.594,E2 -1602.594} C_VEL
LIN {X 0,Y 587.364,Z 527.321,A -85,B 0,C 180,E1 -1605.739,E2 -1605.739} C_VEL
LIN {X 0,Y 587.347,Z 527.316,A -85,B 0,C 180,E1 -1608.866,E2 -1608.866} C_VEL
LIN {X 0,Y 587.372,Z 527.321,A -85,B 0,C 180,E1 -1611.745,E2 -1611.745} C_VEL
LIN {X 0,Y 587.353,Z 527.315,A -85,B 0,C 180,E1 -1614.507,E2 -1614.507} C_VEL
LIN {X 0,Y 587.378,Z 527.315,A -85,B 0,C 180,E1 -1617.257,E2 -1617.257} C_VEL
LIN {X 0,Y 587.382,Z 527.317,A -85,B 0,C 180,E1 -1620,E2 -1620} C_VEL
LIN {X 0,Y 587.378,Z 527.312,A -85,B 0,C 180,E1 -1622.743,E2 -1622.743} C_VEL
LIN {X 0,Y 587.355,Z 527.319,A -85,B 0,C 180,E1 -1625.493,E2 -1625.493} C_VEL
LIN {X 0,Y 587.371,Z 527.316,A -85,B 0,C 180,E1 -1628.255,E2 -1628.255} C_VEL
LIN {X 0,Y 587.347,Z 527.316,A -85,B 0,C 180,E1 -1631.134,E2 -1631.134} C_VEL
LIN {X 0,Y 587.364,Z 527.318,A -85,B 0,C 180,E1 -1634.261,E2 -1634.261} C_VEL
LIN {X 0,Y 587.357,Z 527.318,A -85,B 0,C 180,E1 -1637.406,E2 -1637.406} C_VEL
LIN {X 0,Y 587.324,Z 527.322,A -85,B 0,C 180,E1 -1638.316,E2 -1638.316} C_VEL
LIN {X 0,Y 586.67,Z 527.401,A -85,B 0,C 180,E1 -1638.888,E2 -1638.888} C_VEL
LIN {X 0,Y 583.838,Z 527.76,A -85,B 0,C 180,E1 -1639.816,E2 -1639.816} C_VEL
LIN {X 0,Y 581.428,Z 528.057,A -85,B 0,C 180,E1 -1640.563,E2 -1640.563} C_VEL
LIN {X 0,Y 580.377,Z 528.185,A -85,B 0,C 180,E1 -1641.14,E2 -1641.14} C_VEL
LIN {X 0,Y 580.282,Z 528.197,A -85,B 0,C 180,E1 -1641.335,E2 -1641.335} C_VEL
LIN {X 0,Y 580.301,Z 528.197,A -85,B 0,C 180,E1 -1644.316,E2 -1644.316} C_VEL
LIN {X 0,Y 580.276,Z 528.198,A -85,B 0,C 180,E1 -1646.624,E2 -1646.624} C_VEL
LIN {X 0,Y 580.301,Z 528.194,A -85,B 0,C 180,E1 -1649.31,E2 -1649.31} C_VEL
LIN {X 0,Y 580.297,Z 528.204,A -85,B 0,C 180,E1 -1652.201,E2 -1652.201} C_VEL
LIN {X 0,Y 580.289,Z 528.197,A -85,B 0,C 180,E1 -1654.697,E2 -1654.697} C_VEL
LIN {X 0,Y 580.3,Z 528.194,A -85,B 0,C 180,E1 -1657.269,E2 -1657.269} C_VEL
LIN {X 0,Y 580.298,Z 528.204,A -85,B 0,C 180,E1 -1660.271,E2 -1660.271} C_VEL
LIN {X 0,Y 580.283,Z 528.198,A -85,B 0,C 180,E1 -1662.706,E2 -1662.706} C_VEL
LIN {X 0,Y 580.259,Z 528.201,A -85,B 0,C 180,E1 -1665.611,E2 -1665.611} C_VEL
LIN {X 0,Y 580.28,Z 528.204,A -85,B 0,C 180,E1 -1668.231,E2 -1668.231} C_VEL
LIN {X 0,Y 580.276,Z 528.198,A -85,B 0,C 180,E1 -1670.965,E2 -1670.965} C_VEL
LIN {X 0,Y 580.271,Z 528.199,A -85,B 0,C 180,E1 -1673.596,E2 -1673.596} C_VEL
LIN {X 0,Y 580.321,Z 528.198,A -85,B 0,C 180,E1 -1676.145,E2 -1676.145} C_VEL
LIN {X 0,Y 580.279,Z 528.206,A -85,B 0,C 180,E1 -1678.615,E2 -1678.615} C_VEL
LIN {X 0,Y 580.296,Z 528.198,A -85,B 0,C 180,E1 -1681.024,E2 -1681.024} C_VEL
LIN {X 0,Y 580.295,Z 528.198,A -85,B 0,C 180,E1 -1683.666,E2 -1683.666} C_VEL
LIN {X 0,Y 580.321,Z 528.375,A -85,B 0,C 180,E1 -1684.777,E2 -1684.777} C_VEL
LIN {X 0,Y 581.261,Z 533.124,A -85,B 0,C 180,E1 -1685.438,E2 -1685.438} C_VEL
LIN {X 0,Y 581.084,Z 551.521,A -85,B 0,C 180,E1 -1687.793,E2 -1687.793} C_VEL
LIN {X 0,Y 580.835,Z 573.156,A -85,B 0,C 180,E1 -1690.513,E2 -1690.513} C_VEL
LIN {X 0,Y 580.646,Z 594.144,A -85,B 0,C 180,E1 -1693.112,E2 -1693.112} C_VEL
LIN {X 0,Y 580.464,Z 617.661,A -85,B 0,C 180,E1 -1695.986,E2 -1695.986} C_VEL
LIN {X 0,Y 580.465,Z 620.785,A -85,B 0,C 180,E1 -1696.366,E2 -1696.366} C_VEL
LIN {X 0,Y 580.939,Z 625.654,A -85,B 0,C 180,E1 -1696.444,E2 -1696.444} C_VEL
LIN {X 0,Y 580.803,Z 729.853,A -85,B 0,C 180,E1 -1697.752,E2 -1697.752} C_VEL
LIN {X 0,Y 580.748,Z 743.211,A -85,B 0,C 180,E1 -1698.061,E2 -1698.061} C_VEL
LIN {X 0,Y 580.676,Z 755.362,A -85,B 0,C 180,E1 -1698.48,E2 -1698.48} C_VEL
LIN {X 0,Y 580.597,Z 766.764,A -85,B 0,C 180,E1 -1699.009,E2 -1699.009} C_VEL
LIN {X 0,Y 580.451,Z 778.552,A -85,B 0,C 180,E1 -1699.712,E2 -1699.712} C_VEL
LIN {X 0,Y 580.344,Z 789.057,A -85,B 0,C 180,E1 -1700.502,E2 -1700.502} C_VEL
LIN {X 0,Y 580.302,Z 799.376,A -85,B 0,C 180,E1 -1701.468,E2 -1701.468} C_VEL
LIN {X 0,Y 580.2,Z 808.345,A -85,B 0,C 180,E1 -1702.517,E2 -1702.517} C_VEL
LIN {X 0,Y 580.136,Z 816.001,A -85,B 0,C 180,E1 -1703.637,E2 -1703.637} C_VEL
LIN {X 0,Y 580.086,Z 822.16,A -85,B 0,C 180,E1 -1704.786,E2 -1704.786} C_VEL
LIN {X 0,Y 580.105,Z 826.519,A -85,B 0,C 180,E1 -1705.831,E2 -1705.831} C_VEL
LIN {X 0,Y 580.123,Z 828.82,A -85,B 0,C 180,E1 -1706.527,E2 -1706.527} C_VEL
LIN {X 0,Y 580.043,Z 830.693,A -85,B 0,C 180,E1 -1707.222,E2 -1707.222} C_VEL
LIN {X 0,Y 580.038,Z 832.128,A -85,B 0,C 180,E1 -1707.916,E2 -1707.916} C_VEL
LIN {X 0,Y 580.041,Z 833.753,A -85,B 0,C 180,E1 -1709.305,E2 -1709.305} C_VEL
LIN {X 0,Y 580.038,Z 833.996,A -85,B 0,C 180,E1 -1709.999,E2 -1709.999} C_VEL
LIN {X 0,Y 580.04,Z 833.814,A -85,B 0,C 180,E1 -1710.694,E2 -1710.694} C_VEL
LIN {X 0,Y 580.039,Z 832.272,A -85,B 0,C 180,E1 -1712.083,E2 -1712.083} C_VEL
LIN {X 0,Y 580.044,Z 830.914,A -85,B 0,C 180,E1 -1712.777,E2 -1712.777} C_VEL
LIN {X 0,Y 580.11,Z 828.04,A -85,B 0,C 180,E1 -1713.82,E2 -1713.82} C_VEL
LIN {X 0,Y 580.054,Z 824.142,A -85,B 0,C 180,E1 -1714.865,E2 -1714.865} C_VEL
LIN {X 0,Y 580.162,Z 819.111,A -85,B 0,C 180,E1 -1715.909,E2 -1715.909} C_VEL
LIN {X 0,Y 580.157,Z 812.778,A -85,B 0,C 180,E1 -1716.957,E2 -1716.957} C_VEL
LIN {X 0,Y 580.241,Z 804.875,A -85,B 0,C 180,E1 -1718.006,E2 -1718.006} C_VEL
LIN {X 0,Y 580.304,Z 796.806,A -85,B 0,C 180,E1 -1718.882,E2 -1718.882} C_VEL
LIN {X 0,Y 580.368,Z 786.971,A -85,B 0,C 180,E1 -1719.76,E2 -1719.76} C_VEL
LIN {X 0,Y 580.511,Z 775.915,A -85,B 0,C 180,E1 -1720.55,E2 -1720.55} C_VEL
LIN {X 0,Y 580.614,Z 765.098,A -85,B 0,C 180,E1 -1721.166,E2 -1721.166} C_VEL
LIN {X 0,Y 580.664,Z 752.366,A -85,B 0,C 180,E1 -1721.727,E2 -1721.727} C_VEL
LIN {X 0,Y 580.776,Z 739.281,A -85,B 0,C 180,E1 -1722.137,E2 -1722.137} C_VEL
LIN {X 0,Y 580.805,Z 725.764,A -85,B 0,C 180,E1 -1722.402,E2 -1722.402} C_VEL
LIN {X 0,Y 580.821,Z 624.477,A -85,B 0,C 180,E1 -1723.664,E2 -1723.664} C_VEL
LIN {X 0,Y 580.414,Z 621.531,A -85,B 0,C 180,E1 -1723.724,E2 -1723.724} C_VEL
LIN {X 0,Y 580.571,Z 599.704,A -85,B 0,C 180,E1 -1726.708,E2 -1726.708} C_VEL
LIN {X 0,Y 580.788,Z 577.383,A -85,B 0,C 180,E1 -1729.804,E2 -1729.804} C_VEL
LIN {X 0,Y 580.981,Z 556.375,A -85,B 0,C 180,E1 -1732.773,E2 -1732.773} C_VEL
LIN {X 0,Y 581.231,Z 536.679,A -85,B 0,C 180,E1 -1735.611,E2 -1735.611} C_VEL
LIN {X 0,Y 581.095,Z 531.886,A -85,B 0,C 180,E1 -1736.321,E2 -1736.321} C_VEL
LIN {X 0,Y 580.299,Z 528.204,A -85,B 0,C 180,E1 -1736.913,E2 -1736.913} C_VEL
LIN {X 0,Y 580.287,Z 528.199,A -85,B 0,C 180,E1 -1739.772,E2 -1739.772} C_VEL
LIN {X 0,Y 580.302,Z 528.195,A -85,B 0,C 180,E1 -1742.199,E2 -1742.199} C_VEL
LIN {X 0,Y 580.3,Z 528.197,A -85,B 0,C 180,E1 -1744.694,E2 -1744.694} C_VEL
LIN {X 0,Y 580.297,Z 528.205,A -85,B 0,C 180,E1 -1747.267,E2 -1747.267} C_VEL
LIN {X 0,Y 580.295,Z 528.195,A -85,B 0,C 180,E1 -1750.27,E2 -1750.27} C_VEL
LIN {X 0,Y 580.277,Z 528.198,A -85,B 0,C 180,E1 -1752.705,E2 -1752.705} C_VEL
LIN {X 0,Y 580.268,Z 528.204,A -85,B 0,C 180,E1 -1755.608,E2 -1755.608} C_VEL
LIN {X 0,Y 580.314,Z 528.193,A -85,B 0,C 180,E1 -1758.234,E2 -1758.234} C_VEL
LIN {X 0,Y 580.287,Z 528.2,A -85,B 0,C 180,E1 -1760.965,E2 -1760.965} C_VEL
LIN {X 0,Y 580.291,Z 528.204,A -85,B 0,C 180,E1 -1763.598,E2 -1763.598} C_VEL
LIN {X 0,Y 580.328,Z 528.202,A -85,B 0,C 180,E1 -1764.71,E2 -1764.71} C_VEL
LIN {X 0,Y 580.934,Z 531.723,A -85,B 0,C 180,E1 -1764.768,E2 -1764.768} C_VEL
LIN {X 0,Y 580.759,Z 609.889,A -85,B 0,C 180,E1 -1765.756,E2 -1765.756} C_VEL
LIN {X 0,Y 580.734,Z 622.565,A -85,B 0,C 180,E1 -1766.042,E2 -1766.042} C_VEL
LIN {X 0,Y 580.655,Z 636.08,A -85,B 0,C 180,E1 -1766.509,E2 -1766.509} C_VEL
LIN {X 0,Y 580.501,Z 648.255,A -85,B 0,C 180,E1 -1767.092,E2 -1767.092} C_VEL
LIN {X 0,Y 580.442,Z 658.385,A -85,B 0,C 180,E1 -1767.706,E2 -1767.706} C_VEL
LIN {X 0,Y 580.366,Z 667.971,A -85,B 0,C 180,E1 -1768.416,E2 -1768.416} C_VEL
LIN {X 0,Y 580.305,Z 677.722,A -85,B 0,C 180,E1 -1769.3,E2 -1769.3} C_VEL
LIN {X 0,Y 580.22,Z 687.117,A -85,B 0,C 180,E1 -1770.361,E2 -1770.361} C_VEL
LIN {X 0,Y 580.142,Z 694.558,A -85,B 0,C 180,E1 -1771.411,E2 -1771.411} C_VEL
LIN {X 0,Y 580.101,Z 700.122,A -85,B 0,C 180,E1 -1772.381,E2 -1772.381} C_VEL
LIN {X 0,Y 580.111,Z 704.685,A -85,B 0,C 180,E1 -1773.368,E2 -1773.368} C_VEL
LIN {X 0,Y 580.072,Z 708.794,A -85,B 0,C 180,E1 -1774.525,E2 -1774.525} C_VEL
LIN {X 0,Y 580.022,Z 711.647,A -85,B 0,C 180,E1 -1775.671,E2 -1775.671} C_VEL
LIN {X 0,Y 580.05,Z 713.581,A -85,B 0,C 180,E1 -1777.044,E2 -1777.044} C_VEL
LIN {X 0,Y 580.031,Z 713.982,A -85,B 0,C 180,E1 -1777.938,E2 -1777.938} C_VEL
LIN {X 0,Y 580.054,Z 713.683,A -85,B 0,C 180,E1 -1778.894,E2 -1778.894} C_VEL
LIN {X 0,Y 580.046,Z 712.144,A -85,B 0,C 180,E1 -1780.168,E2 -1780.168} C_VEL
LIN {X 0,Y 580.064,Z 709.661,A -85,B 0,C 180,E1 -1781.277,E2 -1781.277} C_VEL
LIN {X 0,Y 580.083,Z 706.122,A -85,B 0,C 180,E1 -1782.369,E2 -1782.369} C_VEL
LIN {X 0,Y 580.099,Z 701.277,A -85,B 0,C 180,E1 -1783.483,E2 -1783.483} C_VEL
LIN {X 0,Y 580.159,Z 695.398,A -85,B 0,C 180,E1 -1784.543,E2 -1784.543} C_VEL
LIN {X 0,Y 580.216,Z 688.606,A -85,B 0,C 180,E1 -1785.533,E2 -1785.533} C_VEL
LIN {X 0,Y 580.26,Z 680.349,A -85,B 0,C 180,E1 -1786.517,E2 -1786.517} C_VEL
LIN {X 0,Y 580.349,Z 670.112,A -85,B 0,C 180,E1 -1787.498,E2 -1787.498} C_VEL
LIN {X 0,Y 580.415,Z 659.672,A -85,B 0,C 180,E1 -1788.298,E2 -1788.298} C_VEL
LIN {X 0,Y 580.522,Z 649.664,A -85,B 0,C 180,E1 -1788.919,E2 -1788.919} C_VEL
LIN {X 0,Y 580.621,Z 639.004,A -85,B 0,C 180,E1 -1789.451,E2 -1789.451} C_VEL
LIN {X 0,Y 580.702,Z 627.556,A -85,B 0,C 180,E1 -1789.893,E2 -1789.893} C_VEL
LIN {X 0,Y 580.791,Z 614.629,A -85,B 0,C 180,E1 -1790.246,E2 -1790.246} C_VEL
LIN {X 0,Y 580.851,Z 598.896,A -85,B 0,C 180,E1 -1790.489,E2 -1790.489} C_VEL
LIN {X 0,Y 580.823,Z 530.112,A -85,B 0,C 180,E1 -1791.344,E2 -1791.344} C_VEL
LIN {X 0,Y 580.315,Z 528.195,A -85,B 0,C 180,E1 -1791.381,E2 -1791.381} C_VEL
LIN {X 0,Y 580.29,Z 528.197,A -85,B 0,C 180,E1 -1793.742,E2 -1793.742} C_VEL
LIN {X 0,Y 580.27,Z 528.199,A -85,B 0,C 180,E1 -1795.833,E2 -1795.833} C_VEL
LIN {X 0,Y 580.329,Z 528.192,A -85,B 0,C 180,E1 -1797.918,E2 -1797.918} C_VEL
LIN {X 0,Y 580.363,Z 528.198,A -85,B 0,C 180,E1 -1800.694,E2 -1800.694} C_VEL
LIN {X 0,Y 580.282,Z 528.197,A -85,B 0,C 180,E1 -1803.472,E2 -1803.472} C_VEL
LIN {X 0,Y 580.323,Z 528.192,A -85,B 0,C 180,E1 -1805.56,E2 -1805.56} C_VEL
LIN {X 0,Y 580.328,Z 528.195,A -85,B 0,C 180,E1 -1808.356,E2 -1808.356} C_VEL
LIN {X 0,Y 580.322,Z 528.195,A -85,B 0,C 180,E1 -1811.209,E2 -1811.209} C_VEL
LIN {X 0,Y 580.304,Z 528.198,A -85,B 0,C 180,E1 -1814.339,E2 -1814.339} C_VEL
LIN {X 0,Y 580.303,Z 528.202,A -85,B 0,C 180,E1 -1816.915,E2 -1816.915} C_VEL
LIN {X 0,Y 580.298,Z 528.195,A -85,B 0,C 180,E1 -1819.823,E2 -1819.823} C_VEL
LIN {X 0,Y 580.265,Z 528.2,A -85,B 0,C 180,E1 -1822.053,E2 -1822.053} C_VEL
LIN {X 0,Y 580.3,Z 528.2,A -85,B 0,C 180,E1 -1825.08,E2 -1825.08} C_VEL
LIN {X 0,Y 580.311,Z 528.193,A -85,B 0,C 180,E1 -1827.864,E2 -1827.864} C_VEL
LIN {X 0,Y 580.293,Z 528.204,A -85,B 0,C 180,E1 -1830.698,E2 -1830.698} C_VEL
LIN {X 0,Y 580.297,Z 528.197,A -85,B 0,C 180,E1 -1833.318,E2 -1833.318} C_VEL
LIN {X 0,Y 580.32,Z 528.192,A -85,B 0,C 180,E1 -1835.769,E2 -1835.769} C_VEL
LIN {X 0,Y 580.285,Z 528.197,A -85,B 0,C 180,E1 -1838.147,E2 -1838.147} C_VEL
LIN {X 0,Y 580.314,Z 528.203,A -85,B 0,C 180,E1 -1840.842,E2 -1840.842} C_VEL
LIN {X 0,Y 580.285,Z 528.197,A -85,B 0,C 180,E1 -1843.657,E2 -1843.657} C_VEL
LIN {X 0,Y 580.28,Z 528.203,A -85,B 0,C 180,E1 -1846.609,E2 -1846.609} C_VEL
LIN {X 0,Y 580.297,Z 528.201,A -85,B 0,C 180,E1 -1849.158,E2 -1849.158} C_VEL
LIN {X 0,Y 580.287,Z 528.196,A -85,B 0,C 180,E1 -1851.928,E2 -1851.928} C_VEL
LIN {X 0,Y 580.304,Z 528.198,A -85,B 0,C 180,E1 -1854.458,E2 -1854.458} C_VEL
LIN {X 0,Y 580.29,Z 528.205,A -85,B 0,C 180,E1 -1856.976,E2 -1856.976} C_VEL
LIN {X 0,Y 580.3,Z 528.198,A -85,B 0,C 180,E1 -1859.427,E2 -1859.427} C_VEL
LIN {X 0,Y 580.319,Z 528.195,A -85,B 0,C 180,E1 -1862.138,E2 -1862.138} C_VEL
LIN {X 0,Y 580.317,Z 528.299,A -85,B 0,C 180,E1 -1862.894,E2 -1862.894} C_VEL
LIN {X 0,Y 581.662,Z 534.018,A -85,B 0,C 180,E1 -1863.621,E2 -1863.621} C_VEL
LIN {X 0,Y 581.415,Z 557.716,A -85,B 0,C 180,E1 -1866.303,E2 -1866.303} C_VEL
LIN {X 0,Y 581.115,Z 582.931,A -85,B 0,C 180,E1 -1869.099,E2 -1869.099} C_VEL
LIN {X 0,Y 580.837,Z 609.826,A -85,B 0,C 180,E1 -1872.029,E2 -1872.029} C_VEL
LIN {X 0,Y 580.609,Z 635.041,A -85,B 0,C 180,E1 -1874.736,E2 -1874.736} C_VEL
LIN {X 0,Y 580.529,Z 649.75,A -85,B 0,C 180,E1 -1876.301,E2 -1876.301} C_VEL
LIN {X 0,Y 580.987,Z 655.785,A -85,B 0,C 180,E1 -1876.402,E2 -1876.402} C_VEL
LIN {X 0,Y 580.817,Z 759.986,A -85,B 0,C 180,E1 -1877.709,E2 -1877.709} C_VEL
LIN {X 0,Y 580.749,Z 772.481,A -85,B 0,C 180,E1 -1877.996,E2 -1877.996} C_VEL
LIN {X 0,Y 580.66,Z 785.388,A -85,B 0,C 180,E1 -1878.437,E2 -1878.437} C_VEL
LIN {X 0,Y 580.563,Z 797.645,A -85,B 0,C 180,E1 -1879.009,E2 -1879.009} C_VEL
LIN {X 0,Y 580.43,Z 809.213,A -85,B 0,C 180,E1 -1879.713,E2 -1879.713} C_VEL
LIN {X 0,Y 580.341,Z 819.607,A -85,B 0,C 180,E1 -1880.503,E2 -1880.503} C_VEL
LIN {X 0,Y 580.271,Z 828.12,A -85,B 0,C 180,E1 -1881.293,E2 -1881.293} C_VEL
LIN {X 0,Y 580.221,Z 835.966,A -85,B 0,C 180,E1 -1882.169,E2 -1882.169} C_VEL
LIN {X 0,Y 580.154,Z 843.654,A -85,B 0,C 180,E1 -1883.222,E2 -1883.222} C_VEL
LIN {X 0,Y 580.139,Z 850.683,A -85,B 0,C 180,E1 -1884.439,E2 -1884.439} C_VEL
LIN {X 0,Y 580.108,Z 855.374,A -85,B 0,C 180,E1 -1885.484,E2 -1885.484} C_VEL
LIN {X 0,Y 580.123,Z 858.96,A -85,B 0,C 180,E1 -1886.528,E2 -1886.528} C_VEL
LIN {X 0,Y 580.043,Z 860.811,A -85,B 0,C 180,E1 -1887.223,E2 -1887.223} C_VEL
LIN {X 0,Y 580.038,Z 862.202,A -85,B 0,C 180,E1 -1887.917,E2 -1887.917} C_VEL
LIN {X 0,Y 580.04,Z 863.785,A -85,B 0,C 180,E1 -1889.306,E2 -1889.306} C_VEL
LIN {X 0,Y 580.037,Z 864,A -85,B 0,C 180,E1 -1890.001,E2 -1890.001} C_VEL
LIN {X 0,Y 580.047,Z 863.184,A -85,B 0,C 180,E1 -1891.389,E2 -1891.389} C_VEL
LIN {X 0,Y 580.038,Z 862.199,A -85,B 0,C 180,E1 -1892.084,E2 -1892.084} C_VEL
LIN {X 0,Y 580.043,Z 860.807,A -85,B 0,C 180,E1 -1892.778,E2 -1892.778} C_VEL
LIN {X 0,Y 580.11,Z 857.894,A -85,B 0,C 180,E1 -1893.821,E2 -1893.821} C_VEL
LIN {X 0,Y 580.054,Z 853.948,A -85,B 0,C 180,E1 -1894.866,E2 -1894.866} C_VEL
LIN {X 0,Y 580.139,Z 847.874,A -85,B 0,C 180,E1 -1896.085,E2 -1896.085} C_VEL
LIN {X 0,Y 580.185,Z 841.234,A -85,B 0,C 180,E1 -1897.133,E2 -1897.133} C_VEL
LIN {X 0,Y 580.25,Z 832.986,A -85,B 0,C 180,E1 -1898.182,E2 -1898.182} C_VEL
LIN {X 0,Y 580.308,Z 824.533,A -85,B 0,C 180,E1 -1899.059,E2 -1899.059} C_VEL
LIN {X 0,Y 580.417,Z 814.09,A -85,B 0,C 180,E1 -1899.936,E2 -1899.936} C_VEL
LIN {X 0,Y 580.513,Z 803.75,A -85,B 0,C 180,E1 -1900.64,E2 -1900.64} C_VEL
LIN {X 0,Y 580.598,Z 792.23,A -85,B 0,C 180,E1 -1901.265,E2 -1901.265} C_VEL
LIN {X 0,Y 580.707,Z 779.464,A -85,B 0,C 180,E1 -1901.785,E2 -1901.785} C_VEL
LIN {X 0,Y 580.734,Z 766.422,A -85,B 0,C 180,E1 -1902.161,E2 -1902.161} C_VEL
LIN {X 0,Y 580.827,Z 754.055,A -85,B 0,C 180,E1 -1902.381,E2 -1902.381} C_VEL
LIN {X 0,Y 580.815,Z 653.007,A -85,B 0,C 180,E1 -1903.637,E2 -1903.637} C_VEL
LIN {X 0,Y 580.461,Z 650.468,A -85,B 0,C 180,E1 -1903.701,E2 -1903.701} C_VEL
LIN {X 0,Y 580.624,Z 628.33,A -85,B 0,C 180,E1 -1906.345,E2 -1906.345} C_VEL
LIN {X 0,Y 580.852,Z 604.88,A -85,B 0,C 180,E1 -1909.183,E2 -1909.183} C_VEL
LIN {X 0,Y 581.107,Z 581.803,A -85,B 0,C 180,E1 -1912.02,E2 -1912.02} C_VEL
LIN {X 0,Y 581.384,Z 558.373,A -85,B 0,C 180,E1 -1914.956,E2 -1914.956} C_VEL
LIN {X 0,Y 581.708,Z 535.03,A -85,B 0,C 180,E1 -1917.947,E2 -1917.947} C_VEL
LIN {X 0,Y 580.327,Z 528.201,A -85,B 0,C 180,E1 -1918.875,E2 -1918.875} C_VEL
LIN {X 0,Y 580.291,Z 528.2,A -85,B 0,C 180,E1 -1921.385,E2 -1921.385} C_VEL
LIN {X 0,Y 580.322,Z 528.192,A -85,B 0,C 180,E1 -1923.854,E2 -1923.854} C_VEL
LIN {X 0,Y 580.301,Z 528.204,A -85,B 0,C 180,E1 -1926.934,E2 -1926.934} C_VEL
LIN {X 0,Y 580.297,Z 528.195,A -85,B 0,C 180,E1 -1929.933,E2 -1929.933} C_VEL
LIN {X 0,Y 580.279,Z 528.201,A -85,B 0,C 180,E1 -1932.706,E2 -1932.706} C_VEL
LIN {X 0,Y 580.276,Z 528.2,A -85,B 0,C 180,E1 -1935.608,E2 -1935.608} C_VEL
LIN {X 0,Y 580.316,Z 528.191,A -85,B 0,C 180,E1 -1938.234,E2 -1938.234} C_VEL
LIN {X 0,Y 580.291,Z 528.202,A -85,B 0,C 180,E1 -1940.966,E2 -1940.966} C_VEL
LIN {X 0,Y 580.298,Z 528.198,A -85,B 0,C 180,E1 -1943.598,E2 -1943.598} C_VEL
LIN {X 0,Y 580.32,Z 528.192,A -85,B 0,C 180,E1 -1946.145,E2 -1946.145} C_VEL
LIN {X 0,Y 580.282,Z 528.196,A -85,B 0,C 180,E1 -1948.615,E2 -1948.615} C_VEL
LIN {X 0,Y 580.293,Z 528.2,A -85,B 0,C 180,E1 -1951.024,E2 -1951.024} C_VEL
LIN {X 0,Y 580.291,Z 528.199,A -85,B 0,C 180,E1 -1953.666,E2 -1953.666} C_VEL
LIN {X 0,Y 580.3,Z 528.198,A -85,B 0,C 180,E1 -1955.684,E2 -1955.684} C_VEL
LIN {X 0,Y 580.272,Z 528.2,A -85,B 0,C 180,E1 -1957.947,E2 -1957.947} C_VEL
LIN {X 0,Y 580.318,Z 528.193,A -85,B 0,C 180,E1 -1960.914,E2 -1960.914} C_VEL
LIN {X 0,Y 580.279,Z 528.201,A -85,B 0,C 180,E1 -1963.826,E2 -1963.826} C_VEL
LIN {X 0,Y 580.325,Z 528.194,A -85,B 0,C 180,E1 -1965.983,E2 -1965.983} C_VEL
LIN {X 0,Y 580.303,Z 528.193,A -85,B 0,C 180,E1 -1968.827,E2 -1968.827} C_VEL
LIN {X 0,Y 580.335,Z 528.199,A -85,B 0,C 180,E1 -1971.644,E2 -1971.644} C_VEL
LIN {X 0,Y 580.32,Z 528.192,A -85,B 0,C 180,E1 -1974.44,E2 -1974.44} C_VEL
LIN {X 0,Y 580.343,Z 528.19,A -85,B 0,C 180,E1 -1977.224,E2 -1977.224} C_VEL
LIN {X 0,Y 580.351,Z 528.193,A -85,B 0,C 180,E1 -1980,E2 -1980} C_VEL
LIN {X 0,Y 580.343,Z 528.188,A -85,B 0,C 180,E1 -1982.777,E2 -1982.777} C_VEL
LIN {X 0,Y 580.322,Z 528.196,A -85,B 0,C 180,E1 -1985.56,E2 -1985.56} C_VEL
LIN {X 0,Y 580.334,Z 528.192,A -85,B 0,C 180,E1 -1988.356,E2 -1988.356} C_VEL
LIN {X 0,Y 580.299,Z 528.195,A -85,B 0,C 180,E1 -1991.191,E2 -1991.191} C_VEL
LIN {X 0,Y 580.325,Z 528.199,A -85,B 0,C 180,E1 -1994.017,E2 -1994.017} C_VEL
LIN {X 0,Y 580.311,Z 528.192,A -85,B 0,C 180,E1 -1996.914,E2 -1996.914} C_VEL
LIN {X 0,Y 580.304,Z 528.2,A -85,B 0,C 180,E1 -1999.822,E2 -1999.822} C_VEL
LIN {X 0,Y 580.282,Z 528.197,A -85,B 0,C 180,E1 -2001.335,E2 -2001.335} C_VEL
LIN {X 0,Y 579.586,Z 528.293,A -85,B 0,C 180,E1 -2001.914,E2 -2001.914} C_VEL
LIN {X 0,Y 576.71,Z 528.648,A -85,B 0,C 180,E1 -2002.854,E2 -2002.854} C_VEL
LIN {X 0,Y 574.316,Z 528.945,A -85,B 0,C 180,E1 -2003.61,E2 -2003.61} C_VEL
LIN {X 0,Y 573.317,Z 529.069,A -85,B 0,C 180,E1 -2004.194,E2 -2004.194} C_VEL
LIN {X 0,Y 573.251,Z 529.073,A -85,B 0,C 180,E1 -2004.392,E2 -2004.392} C_VEL
